// TwinCAT 3 PLC project IoT_OPCUA
// ProgramVersion: 3.1.4023.0
// libraries:
//   Tc2_EtherCAT, * (Beckhoff Automation GmbH)
//   Tc2_MDP, * (Beckhoff Automation GmbH)
//   Tc2_ModbusSrv, * (Beckhoff Automation GmbH)
//   Tc2_Standard, * (Beckhoff Automation GmbH)
//   Tc2_System, * (Beckhoff Automation GmbH)
//   Tc2_Utilities, * (Beckhoff Automation GmbH)
//   Tc3_IPCDiag, * (Beckhoff Automation GmbH)
//   Tc3_Module, * (Beckhoff Automation GmbH)
//   BASIC,3.31,OSCAT
//   Tc2_OpcUa,3.3.2.0,Beckhoff Automation GmbH
//   VisuSymbols,3.5.10.0,System
// project tree:
//   / Class Diagram.TcCD (not stored), GlobalTextList.TcGTLO, PlcTask_10ms.TcTTO, PlcTask_500us.TcTTO, Task_1ms.TcTTO, Visualization Manager.TcVMO (not stored)
//   DUTs/ AirValveSimSignals.TcDUT, ElectrDataModbusTCP.TcDUT, ElectrDataEthCAT.TcDUT
//   DUTs/DataModels/ DriveState_DataModel.TcDUT, ElectrDevicePeriodicOper_DataModel.TcDUT, ElectrDeviceContOper_DataModel.TcDUT, SingleSensor_DataModel.TcDUT, SingleState_DataModel.TcDUT, ValveTravelTime_DataModel.TcDUT, VibAccelarationDataModel.TcDUT
//   GVLs/ GVL_const.TcGVL, GVL_SW.TcGVL, GVL_HW.TcGVL, GVL_Visu.TcGVL
//   POUs/EL3443/EL3443/DUTs/ E_EL3443_Phase.TcDUT, E_EL3443_Total.TcDUT, ST_EL3443_MUX_REAL.TcDUT, ST_EL3443_MUX_ULINT.TcDUT, ST_EL3443_StatusLx.TcDUT, ST_EL3443_StatusTotal.TcDUT, ST_EL3443_VariantLx.TcDUT, ST_EL3443_VariantTotal.TcDUT, ST_EL3443_VariantValues.TcDUT
//   POUs/EL3443/EL3443/ FB_EL3443.TcPOU (not stored)
//   POUs/EL3443/EL3443_DPM/DUTs/ E_EL3443_DPM_Phase.TcDUT, E_EL3443_DPM_Total.TcDUT, ST_EL3443_DPM_MUX_REAL.TcDUT, ST_EL3443_DPM_MUX_ULINT.TcDUT, ST_EL3443_DPM_StatusLx.TcDUT, ST_EL3443_DPM_StatusTotal.TcDUT, ST_EL3443_DPM_VariantLx.TcDUT, ST_EL3443_DPM_VariantTotal.TcDUT, ST_EL3443_DPM_VariantValues.TcDUT
//   POUs/EL3443/EL3443_DPM/ FB_EL3443_DPM.TcPOU
//   POUs/FB/Generic/ CheckLineProducing.TcPOU, PartsPerMinHistorical.TcPOU, PartsPerMinInstant.TcPOU, PartsPerMinInstant2.TcPOU, ReadMemoryUsage.TcPOU, Valve_Signal_Sim.TcPOU, TONR.TcPOU, UnixTimestamp.TcPOU, ValueChangeDetector.TcPOU
//   POUs/FB/ModbusTCP/ ReadMBSentron_PAC1200.TcPOU
//   POUs/FB/OPC_UA/ ElectricalDevicePeriodicOper.TcPOU, ElectricalDeviceContOper.TcPOU, GenericSensor.TcPOU, GenericState.TcPOU, Valve2Cmd2FB.TcPOU, VibrationSensor.TcPOU
//   POUs/FC/ AI_Scale.TcPOU
//   POUs/PRG_10ms/ PRG_06_ElectricalMonitoring.TcPOU, PRG_04_AirValveAnalytics.TcPOU, PRG_05_ElectricalAnalytics.TcPOU, PRG_01_MAIN.TcPOU, PRG_09_PlcDiagnostic.TcPOU, PRG_08_ProductionStatistics.TcPOU, PRG_10_TempHumidAnalytics.TcPOU, PRG_11_AirFlowAnalytics.TcPOU, PRG_12_OilContaminationAnalytics.TcPOU, Simulation.TcPOU, PRG_02_DataMapping.TcPOU, PRG_07_LineState.TcPOU, PRG_03_VibrationAnalytics.TcPOU
//   POUs/PRG_1ms/ Main_T1ms.TcPOU, TimeStamp.TcPOU
//   POUs/PRG_500us/ Main_500us.TcPOU
//   VISU/ TextList1.TcTLO, Visualization1.TcVIS
// real-time tasks:
//   TASK PlcTask_10ms: cycle T#10ms, priority 20, ADS port 350
//   TASK Task_1ms: cycle T#1ms, priority 1, ADS port 351
//   TASK ProfiNET: cycle T#2ms, priority 2, ADS port 301
//   TASK PlcTask_500us: cycle T#500us, priority 23, ADS port 354
// I/O:
//   DEVICE Device1 (Profinet Device) (disabled), AmsNetId 192.168.149.130.2.1
//     profinet-io-device [Beckhoff Automation TwinCAT PLC PROFINET I/O Device with I/Os, V2.32, 1 port diagnostic supported TwinCAT PN Device]
//       modules: Term 1 (DAP Module), Term 2 (32 Word Output), Term 3 (32 DWord Output), Term 4 (10 Float32 Output), Term 5 (10 Float32 Input)
//   DEVICE Device2 (EtherCAT) (disabled), AmsNetId 192.168.149.130.3.1
//     ElectricalCabinet [EK1100 EtherCAT Coupler (2A E-Bus)]
//       Term_1 (EL3443) [EL3443 3Ch. Power Measuring]
//       Term_2 (EL3443) [EL3443 3Ch. Power Measuring]
//       Term_3 (EL3152) [EL3152 2Ch. Ana Input 4-20mA]
//       Term_4 (EL6601) [EL6601 1 Port Switch (Ethernet, CoE)]
//       Term_99 (EL9011) [EL9011 End Terminal]
//     IO_LinkNode1 (EP6228-0022) [EP6228-0022 (IO Link Master)]
//       modules: Module 1 (DeviceState Inputs Device), Module 2 (DeviceState Inputs), IoLinkNode1_Ch1 (IO-Link Slave), IoLinkNode1_Ch2 (IO-Link Slave), IoLinkNode1_Ch3 (IO-Link Slave), IoLinkNode1_Ch4 (IO-Link Slave), IoLinkNode1_Ch5 (IO-Link Slave), IoLinkNode1_Ch6 (IO-Link Slave), Module 9 (empty), Module 10 (empty)
//     IO_LinkNode2 (EP6224-2022) [EP6224-2022 (IO Link Master)]
//       modules: Module 1 (DeviceState Inputs Device), Module 2 (DeviceState Inputs), IoLinkNode2_Ch1 (IO-Link Slave), IoLinkNode2_Ch2 (IO-Link Slave), IoLinkNode2_Ch3 (IO-Link Slave), IoLinkNode2_Ch4 (IO-Link Slave)
//   DEVICE Device 3 (USB) (disabled)
//     Box 2 (C9900-L100 License-Key-USB-Stick)
// variable links:
//   IoT_OPCUA/IoT_OPCUA Instance <-> Device1 (Profinet Device)/profinet-io-device
//     PlcTask_10ms Inputs/GVL_HW.PnIoDevice_10Real_In <-> API/Term 4 (10 Float32 Output)/Subterm 6 (10 Float32 Output)/Inputs/1 Float32 Output[0]
//     PlcTask_10ms Inputs/GVL_HW.PnIoDevice_10Real_In @bit {32..288 step 32} <-> API/Term 4 (10 Float32 Output)/Subterm 6 (10 Float32 Output)/Inputs/1 Float32 Output[{1..9}]  (9 links)
//     PlcTask_10ms Inputs/GVL_HW.PnIoDevice_32DWord_In <-> API/Term 3 (32 DWord Output)/Subterm 5 (32 DWord Output)/Inputs/1 DWord Output[0]
//     PlcTask_10ms Inputs/GVL_HW.PnIoDevice_32DWord_In @bit {32..992 step 32} <-> API/Term 3 (32 DWord Output)/Subterm 5 (32 DWord Output)/Inputs/1 DWord Output[{1..31}]  (31 links)
//     PlcTask_10ms Inputs/GVL_HW.PnIoDevice_32Word_In <-> API/Term 2 (32 Word Output)/Subterm 4 (32 Word Output)/Inputs/1 Word Output[0]
//     PlcTask_10ms Inputs/GVL_HW.PnIoDevice_32Word_In @bit {16..496 step 16} <-> API/Term 2 (32 Word Output)/Subterm 4 (32 Word Output)/Inputs/1 Word Output[{1..31}]  (31 links)
//     PlcTask_10ms Outputs/GVL_HW.PnIoDevice_10Real_Out <-> API/Term 5 (10 Float32 Input)/Subterm 7 (10 Float32 Input)/Outputs/1 Float32 Input[0]
//     PlcTask_10ms Outputs/GVL_HW.PnIoDevice_10Real_Out @bit {32..288 step 32} <-> API/Term 5 (10 Float32 Input)/Subterm 7 (10 Float32 Input)/Outputs/1 Float32 Input[{1..9}]  (9 links)
//   IoT_OPCUA/IoT_OPCUA Instance <-> Device2 (EtherCAT)/ElectricalCabinet/Term_1 (EL3443)
//     PlcTask_500us Inputs/Main_500us.ElectricalDevice1.stEL3443_IO.MDP5001_341_Input/MDP5001_341_L1_Basic_Current <-> L1 Basic/Current
//     PlcTask_500us Inputs/Main_500us.ElectricalDevice1.stEL3443_IO.MDP5001_341_Input/MDP5001_341_L2_Basic_Current <-> L2 Basic/Current
//     PlcTask_500us Inputs/Main_500us.ElectricalDevice1.stEL3443_IO.MDP5001_341_Input/MDP5001_341_L3_Basic_Current <-> L3 Basic/Current
//     PlcTask_500us Inputs/Main_500us.ElectricalDevice1.stEL3443_IO.MDP5001_341_Input/MDP5001_341_L1_Basic_Voltage <-> L1 Basic/Voltage
//     PlcTask_500us Inputs/Main_500us.ElectricalDevice1.stEL3443_IO.MDP5001_341_Input/MDP5001_341_L2_Basic_Voltage <-> L2 Basic/Voltage
//     PlcTask_500us Inputs/Main_500us.ElectricalDevice1.stEL3443_IO.MDP5001_341_Input/MDP5001_341_L3_Basic_Voltage <-> L3 Basic/Voltage
//     PlcTask_500us Inputs/Main_500us.ElectricalDevice1.stEL3443_IO.MDP5001_341_Input/MDP5001_341_L1_Power_Active_Power <-> L1 Power/Active Power
//     PlcTask_500us Inputs/Main_500us.ElectricalDevice1.stEL3443_IO.MDP5001_341_Input/MDP5001_341_L2_Power_Active_Power <-> L2 Power/Active Power
//     PlcTask_500us Inputs/Main_500us.ElectricalDevice1.stEL3443_IO.MDP5001_341_Input/MDP5001_341_L3_Power_Active_Power <-> L3 Power/Active Power
//     PlcTask_500us Inputs/Main_500us.ElectricalDevice1.stEL3443_IO.MDP5001_341_Input/MDP5001_341_L1_Power_Apparent_Power <-> L1 Power/Apparent Power
//     PlcTask_500us Inputs/Main_500us.ElectricalDevice1.stEL3443_IO.MDP5001_341_Input/MDP5001_341_L2_Power_Apparent_Power <-> L2 Power/Apparent Power
//     PlcTask_500us Inputs/Main_500us.ElectricalDevice1.stEL3443_IO.MDP5001_341_Input/MDP5001_341_L3_Power_Apparent_Power <-> L3 Power/Apparent Power
//     PlcTask_500us Inputs/Main_500us.ElectricalDevice1.stEL3443_IO.MDP5001_341_Input/MDP5001_341_L1_Power_Power_Factor <-> L1 Power/Power Factor
//     PlcTask_500us Inputs/Main_500us.ElectricalDevice1.stEL3443_IO.MDP5001_341_Input/MDP5001_341_L2_Power_Power_Factor <-> L2 Power/Power Factor
//     PlcTask_500us Inputs/Main_500us.ElectricalDevice1.stEL3443_IO.MDP5001_341_Input/MDP5001_341_L3_Power_Power_Factor <-> L3 Power/Power Factor
//     PlcTask_500us Inputs/Main_500us.ElectricalDevice1.stEL3443_IO.MDP5001_341_Input/MDP5001_341_L1_Power_Reactive_Power <-> L1 Power/Reactive Power
//     PlcTask_500us Inputs/Main_500us.ElectricalDevice1.stEL3443_IO.MDP5001_341_Input/MDP5001_341_L2_Power_Reactive_Power <-> L2 Power/Reactive Power
//     PlcTask_500us Inputs/Main_500us.ElectricalDevice1.stEL3443_IO.MDP5001_341_Input/MDP5001_341_L3_Power_Reactive_Power <-> L3 Power/Reactive Power
//     PlcTask_500us Inputs/Main_500us.ElectricalDevice1.stEL3443_IO.MDP5001_341_Input/MDP5001_341_L1_Status_Current_Guard_Error <-> L1 Status/Current Guard Error
//     PlcTask_500us Inputs/Main_500us.ElectricalDevice1.stEL3443_IO.MDP5001_341_Input/MDP5001_341_L2_Status_Current_Guard_Error <-> L2 Status/Current Guard Error
//     PlcTask_500us Inputs/Main_500us.ElectricalDevice1.stEL3443_IO.MDP5001_341_Input/MDP5001_341_L3_Status_Current_Guard_Error <-> L3 Status/Current Guard Error
//     PlcTask_500us Inputs/Main_500us.ElectricalDevice1.stEL3443_IO.MDP5001_341_Input/MDP5001_341_L1_Status_Current_Guard_Warning <-> L1 Status/Current Guard Warning
//     PlcTask_500us Inputs/Main_500us.ElectricalDevice1.stEL3443_IO.MDP5001_341_Input/MDP5001_341_L2_Status_Current_Guard_Warning <-> L2 Status/Current Guard Warning
//     PlcTask_500us Inputs/Main_500us.ElectricalDevice1.stEL3443_IO.MDP5001_341_Input/MDP5001_341_L3_Status_Current_Guard_Warning <-> L3 Status/Current Guard Warning
//     PlcTask_500us Inputs/Main_500us.ElectricalDevice1.stEL3443_IO.MDP5001_341_Input/MDP5001_341_L1_Status_Inaccurate_Current <-> L1 Status/Inaccurate Current
//     PlcTask_500us Inputs/Main_500us.ElectricalDevice1.stEL3443_IO.MDP5001_341_Input/MDP5001_341_L2_Status_Inaccurate_Current <-> L2 Status/Inaccurate Current
//     PlcTask_500us Inputs/Main_500us.ElectricalDevice1.stEL3443_IO.MDP5001_341_Input/MDP5001_341_L3_Status_Inaccurate_Current <-> L3 Status/Inaccurate Current
//     PlcTask_500us Inputs/Main_500us.ElectricalDevice1.stEL3443_IO.MDP5001_341_Input/MDP5001_341_L1_Status_Inaccurate_Voltage <-> L1 Status/Inaccurate Voltage
//     PlcTask_500us Inputs/Main_500us.ElectricalDevice1.stEL3443_IO.MDP5001_341_Input/MDP5001_341_L2_Status_Inaccurate_Voltage <-> L2 Status/Inaccurate Voltage
//     PlcTask_500us Inputs/Main_500us.ElectricalDevice1.stEL3443_IO.MDP5001_341_Input/MDP5001_341_L3_Status_Inaccurate_Voltage <-> L3 Status/Inaccurate Voltage
//     PlcTask_500us Inputs/Main_500us.ElectricalDevice1.stEL3443_IO.MDP5001_341_Input/MDP5001_341_L1_Status_Overcurrent <-> L1 Status/Overcurrent
//     PlcTask_500us Inputs/Main_500us.ElectricalDevice1.stEL3443_IO.MDP5001_341_Input/MDP5001_341_L2_Status_Overcurrent <-> L2 Status/Overcurrent
//     PlcTask_500us Inputs/Main_500us.ElectricalDevice1.stEL3443_IO.MDP5001_341_Input/MDP5001_341_L3_Status_Overcurrent <-> L3 Status/Overcurrent
//     PlcTask_500us Inputs/Main_500us.ElectricalDevice1.stEL3443_IO.MDP5001_341_Input/MDP5001_341_L1_Status_Overvoltage <-> L1 Status/Overvoltage
//     PlcTask_500us Inputs/Main_500us.ElectricalDevice1.stEL3443_IO.MDP5001_341_Input/MDP5001_341_L2_Status_Overvoltage <-> L2 Status/Overvoltage
//     PlcTask_500us Inputs/Main_500us.ElectricalDevice1.stEL3443_IO.MDP5001_341_Input/MDP5001_341_L3_Status_Overvoltage <-> L3 Status/Overvoltage
//     PlcTask_500us Inputs/Main_500us.ElectricalDevice1.stEL3443_IO.MDP5001_341_Input/MDP5001_341_L1_Status_TxPDO_Toggle <-> L1 Status/TxPDO Toggle
//     PlcTask_500us Inputs/Main_500us.ElectricalDevice1.stEL3443_IO.MDP5001_341_Input/MDP5001_341_L2_Status_TxPDO_Toggle <-> L2 Status/TxPDO Toggle
//     PlcTask_500us Inputs/Main_500us.ElectricalDevice1.stEL3443_IO.MDP5001_341_Input/MDP5001_341_L3_Status_TxPDO_Toggle <-> L3 Status/TxPDO Toggle
//     PlcTask_500us Inputs/Main_500us.ElectricalDevice1.stEL3443_IO.MDP5001_341_Input/MDP5001_341_L1_Status_Voltage_Guard_Error <-> L1 Status/Voltage Guard Error
//     PlcTask_500us Inputs/Main_500us.ElectricalDevice1.stEL3443_IO.MDP5001_341_Input/MDP5001_341_L2_Status_Voltage_Guard_Error <-> L2 Status/Voltage Guard Error
//     PlcTask_500us Inputs/Main_500us.ElectricalDevice1.stEL3443_IO.MDP5001_341_Input/MDP5001_341_L3_Status_Voltage_Guard_Error <-> L3 Status/Voltage Guard Error
//     PlcTask_500us Inputs/Main_500us.ElectricalDevice1.stEL3443_IO.MDP5001_341_Input/MDP5001_341_L1_Status_Voltage_Guard_Warning <-> L1 Status/Voltage Guard Warning
//     PlcTask_500us Inputs/Main_500us.ElectricalDevice1.stEL3443_IO.MDP5001_341_Input/MDP5001_341_L2_Status_Voltage_Guard_Warning <-> L2 Status/Voltage Guard Warning
//     PlcTask_500us Inputs/Main_500us.ElectricalDevice1.stEL3443_IO.MDP5001_341_Input/MDP5001_341_L3_Status_Voltage_Guard_Warning <-> L3 Status/Voltage Guard Warning
//     PlcTask_500us Inputs/Main_500us.ElectricalDevice1.stEL3443_IO.MDP5001_341_Input/MDP5001_341_L1_Status_Voltage_Sign_Bit <-> L1 Status/Voltage Sign Bit
//     PlcTask_500us Inputs/Main_500us.ElectricalDevice1.stEL3443_IO.MDP5001_341_Input/MDP5001_341_L2_Status_Voltage_Sign_Bit <-> L2 Status/Voltage Sign Bit
//     PlcTask_500us Inputs/Main_500us.ElectricalDevice1.stEL3443_IO.MDP5001_341_Input/MDP5001_341_L3_Status_Voltage_Sign_Bit <-> L3 Status/Voltage Sign Bit
//     PlcTask_500us Inputs/Main_500us.ElectricalDevice1.stEL3443_IO.MDP5001_341_Input/MDP5001_341_L1_Timing_Voltage_Last_Zero_Crossing <-> L1 Timing/Voltage Last Zero Crossing
//     PlcTask_500us Inputs/Main_500us.ElectricalDevice1.stEL3443_IO.MDP5001_341_Input/MDP5001_341_L2_Timing_Voltage_Last_Zero_Crossing <-> L2 Timing/Voltage Last Zero Crossing
//     PlcTask_500us Inputs/Main_500us.ElectricalDevice1.stEL3443_IO.MDP5001_341_Input/MDP5001_341_L3_Timing_Voltage_Last_Zero_Crossing <-> L3 Timing/Voltage Last Zero Crossing
//     PlcTask_500us Inputs/Main_500us.ElectricalDevice1.stEL3443_IO.MDP5001_341_Input/MDP5001_341_Total_Basic_Calculated_Neutral_Line_Current <-> Total Basic/Calculated Neutral Line Current
//     PlcTask_500us Inputs/Main_500us.ElectricalDevice1.stEL3443_IO.MDP5001_341_Input/MDP5001_341_Total_Basic_Frequency <-> Total Basic/Frequency
//     PlcTask_500us Inputs/Main_500us.ElectricalDevice1.stEL3443_IO.MDP5001_341_Input/MDP5001_341_Total_Basic_Power_Factor <-> Total Basic/Power Factor
//     PlcTask_500us Inputs/Main_500us.ElectricalDevice1.stEL3443_IO.MDP5001_341_Input/MDP5001_341_Total_Status_Active_Power_Guard_Error <-> Total Status/Active Power Guard Error
//     PlcTask_500us Inputs/Main_500us.ElectricalDevice1.stEL3443_IO.MDP5001_341_Input/MDP5001_341_Total_Status_Active_Power_Guard_Warning <-> Total Status/Active Power Guard Warning
//     PlcTask_500us Inputs/Main_500us.ElectricalDevice1.stEL3443_IO.MDP5001_341_Input/MDP5001_341_Total_Status_Apparent_Power_Guard_Error <-> Total Status/Apparent Power Guard Error
//     PlcTask_500us Inputs/Main_500us.ElectricalDevice1.stEL3443_IO.MDP5001_341_Input/MDP5001_341_Total_Status_Apparent_Power_Guard_Warning <-> Total Status/Apparent Power Guard Warning
//     PlcTask_500us Inputs/Main_500us.ElectricalDevice1.stEL3443_IO.MDP5001_341_Input/MDP5001_341_Total_Status_Frequency_Guard_Error <-> Total Status/Frequency Guard Error
//     PlcTask_500us Inputs/Main_500us.ElectricalDevice1.stEL3443_IO.MDP5001_341_Input/MDP5001_341_Total_Status_Frequency_Guard_Warning <-> Total Status/Frequency Guard Warning
//     PlcTask_500us Inputs/Main_500us.ElectricalDevice1.stEL3443_IO.MDP5001_341_Input/MDP5001_341_Total_Status_Grid_Direction <-> Total Status/Grid Direction
//     PlcTask_500us Inputs/Main_500us.ElectricalDevice1.stEL3443_IO.MDP5001_341_Input/MDP5001_341_Total_Status_Neutral_Current_Guard_Error <-> Total Status/Neutral Current Guard Error
//     PlcTask_500us Inputs/Main_500us.ElectricalDevice1.stEL3443_IO.MDP5001_341_Input/MDP5001_341_Total_Status_Neutral_Current_Guard_Warning <-> Total Status/Neutral Current Guard Warning
//     PlcTask_500us Inputs/Main_500us.ElectricalDevice1.stEL3443_IO.MDP5001_341_Input/MDP5001_341_Total_Status_Power_Quality_Factor <-> Total Status/Power Quality Factor
//     PlcTask_500us Inputs/Main_500us.ElectricalDevice1.stEL3443_IO.MDP5001_341_Input/MDP5001_341_Total_Status_Power_Quality_Guard_Error <-> Total Status/Power Quality Guard Error
//     PlcTask_500us Inputs/Main_500us.ElectricalDevice1.stEL3443_IO.MDP5001_341_Input/MDP5001_341_Total_Status_Power_Quality_Guard_Warning <-> Total Status/Power Quality Guard Warning
//     PlcTask_500us Inputs/Main_500us.ElectricalDevice1.stEL3443_IO.MDP5001_341_Input/MDP5001_341_Total_Status_System_State <-> Total Status/System State
//     PlcTask_500us Inputs/Main_500us.ElectricalDevice1.stEL3443_IO.MDP5001_341_Input/MDP5001_341_Total_Status_TxPDO_State <-> Total Status/TxPDO State
//     PlcTask_500us Inputs/Main_500us.ElectricalDevice1.stEL3443_IO.MDP5001_341_Input/MDP5001_341_Total_Status_TxPDO_Toggle <-> Total Status/TxPDO Toggle
//     PlcTask_500us Inputs/Main_500us.ElectricalDevice1.stEL3443_IO.MDP5001_341_Input/MDP5001_341_Total_Variant_Value_In_Index_1_REAL <-> Total Variant Value In/Index 1 REAL
//     PlcTask_500us Inputs/Main_500us.ElectricalDevice1.stEL3443_IO.MDP5001_341_Input/MDP5001_341_Total_Variant_Value_In_Index_2_REAL <-> Total Variant Value In/Index 2 REAL
//     PlcTask_500us Inputs/Main_500us.ElectricalDevice1.stEL3443_IO.MDP5001_341_Input/MDP5001_341_Total_Variant_Value_In_Index_3_REAL <-> Total Variant Value In/Index 3 REAL
//     PlcTask_500us Inputs/Main_500us.ElectricalDevice1.stEL3443_IO.MDP5001_341_Input/MDP5001_341_Total_Variant_Value_In_Index_4_ULINT <-> Total Variant Value In/Index 4 ULINT
//     PlcTask_500us Inputs/Main_500us.ElectricalDevice1.stEL3443_IO.MDP5001_341_Input/MDP5001_341_Total_Variant_Value_In_TxPDO_Toggle <-> Total Variant Value In/TxPDO Toggle
//     PlcTask_500us Inputs/Main_500us.ElectricalDevice1.stEL3443_IO.MDP5001_341_Input/MDP5001_341_Total_Variant_Value_In_Value_1_REAL <-> Total Variant Value In/Value 1 REAL
//     PlcTask_500us Inputs/Main_500us.ElectricalDevice1.stEL3443_IO.MDP5001_341_Input/MDP5001_341_Total_Variant_Value_In_Value_2_REAL <-> Total Variant Value In/Value 2 REAL
//     PlcTask_500us Inputs/Main_500us.ElectricalDevice1.stEL3443_IO.MDP5001_341_Input/MDP5001_341_Total_Variant_Value_In_Value_3_REAL <-> Total Variant Value In/Value 3 REAL
//     PlcTask_500us Inputs/Main_500us.ElectricalDevice1.stEL3443_IO.MDP5001_341_Input/MDP5001_341_Total_Variant_Value_In_Value_4_ULINT <-> Total Variant Value In/Value 4 ULINT
//     PlcTask_500us Outputs/Main_500us.ElectricalDevice1.stEL3443_IO.MDP5001_341_Output/MDP5001_341_Total_Variant_Value_Out_Index_1_REAL <-> Total Variant Value Out/Index 1 REAL
//     PlcTask_500us Outputs/Main_500us.ElectricalDevice1.stEL3443_IO.MDP5001_341_Output/MDP5001_341_Total_Variant_Value_Out_Index_2_REAL <-> Total Variant Value Out/Index 2 REAL
//     PlcTask_500us Outputs/Main_500us.ElectricalDevice1.stEL3443_IO.MDP5001_341_Output/MDP5001_341_Total_Variant_Value_Out_Index_3_REAL <-> Total Variant Value Out/Index 3 REAL
//     PlcTask_500us Outputs/Main_500us.ElectricalDevice1.stEL3443_IO.MDP5001_341_Output/MDP5001_341_Total_Variant_Value_Out_Index_4_ULINT <-> Total Variant Value Out/Index 4 ULINT
//   IoT_OPCUA/IoT_OPCUA Instance <-> Device2 (EtherCAT)/ElectricalCabinet/Term_2 (EL3443)
//     PlcTask_500us Inputs/Main_500us.ElectricalDevice2.stEL3443_IO.MDP5001_341_Input/MDP5001_341_L1_Basic_Current <-> L1 Basic/Current
//     PlcTask_500us Inputs/Main_500us.ElectricalDevice2.stEL3443_IO.MDP5001_341_Input/MDP5001_341_L2_Basic_Current <-> L2 Basic/Current
//     PlcTask_500us Inputs/Main_500us.ElectricalDevice2.stEL3443_IO.MDP5001_341_Input/MDP5001_341_L3_Basic_Current <-> L3 Basic/Current
//     PlcTask_500us Inputs/Main_500us.ElectricalDevice2.stEL3443_IO.MDP5001_341_Input/MDP5001_341_L1_Basic_Voltage <-> L1 Basic/Voltage
//     PlcTask_500us Inputs/Main_500us.ElectricalDevice2.stEL3443_IO.MDP5001_341_Input/MDP5001_341_L2_Basic_Voltage <-> L2 Basic/Voltage
//     PlcTask_500us Inputs/Main_500us.ElectricalDevice2.stEL3443_IO.MDP5001_341_Input/MDP5001_341_L3_Basic_Voltage <-> L3 Basic/Voltage
//     PlcTask_500us Inputs/Main_500us.ElectricalDevice2.stEL3443_IO.MDP5001_341_Input/MDP5001_341_L1_Power_Active_Power <-> L1 Power/Active Power
//     PlcTask_500us Inputs/Main_500us.ElectricalDevice2.stEL3443_IO.MDP5001_341_Input/MDP5001_341_L2_Power_Active_Power <-> L2 Power/Active Power
//     PlcTask_500us Inputs/Main_500us.ElectricalDevice2.stEL3443_IO.MDP5001_341_Input/MDP5001_341_L3_Power_Active_Power <-> L3 Power/Active Power
//     PlcTask_500us Inputs/Main_500us.ElectricalDevice2.stEL3443_IO.MDP5001_341_Input/MDP5001_341_L1_Power_Apparent_Power <-> L1 Power/Apparent Power
//     PlcTask_500us Inputs/Main_500us.ElectricalDevice2.stEL3443_IO.MDP5001_341_Input/MDP5001_341_L2_Power_Apparent_Power <-> L2 Power/Apparent Power
//     PlcTask_500us Inputs/Main_500us.ElectricalDevice2.stEL3443_IO.MDP5001_341_Input/MDP5001_341_L3_Power_Apparent_Power <-> L3 Power/Apparent Power
//     PlcTask_500us Inputs/Main_500us.ElectricalDevice2.stEL3443_IO.MDP5001_341_Input/MDP5001_341_L1_Power_Power_Factor <-> L1 Power/Power Factor
//     PlcTask_500us Inputs/Main_500us.ElectricalDevice2.stEL3443_IO.MDP5001_341_Input/MDP5001_341_L2_Power_Power_Factor <-> L2 Power/Power Factor
//     PlcTask_500us Inputs/Main_500us.ElectricalDevice2.stEL3443_IO.MDP5001_341_Input/MDP5001_341_L3_Power_Power_Factor <-> L3 Power/Power Factor
//     PlcTask_500us Inputs/Main_500us.ElectricalDevice2.stEL3443_IO.MDP5001_341_Input/MDP5001_341_L1_Power_Reactive_Power <-> L1 Power/Reactive Power
//     PlcTask_500us Inputs/Main_500us.ElectricalDevice2.stEL3443_IO.MDP5001_341_Input/MDP5001_341_L2_Power_Reactive_Power <-> L2 Power/Reactive Power
//     PlcTask_500us Inputs/Main_500us.ElectricalDevice2.stEL3443_IO.MDP5001_341_Input/MDP5001_341_L3_Power_Reactive_Power <-> L3 Power/Reactive Power
//     PlcTask_500us Inputs/Main_500us.ElectricalDevice2.stEL3443_IO.MDP5001_341_Input/MDP5001_341_L1_Status_Current_Guard_Error <-> L1 Status/Current Guard Error
//     PlcTask_500us Inputs/Main_500us.ElectricalDevice2.stEL3443_IO.MDP5001_341_Input/MDP5001_341_L2_Status_Current_Guard_Error <-> L2 Status/Current Guard Error
//     PlcTask_500us Inputs/Main_500us.ElectricalDevice2.stEL3443_IO.MDP5001_341_Input/MDP5001_341_L3_Status_Current_Guard_Error <-> L3 Status/Current Guard Error
//     PlcTask_500us Inputs/Main_500us.ElectricalDevice2.stEL3443_IO.MDP5001_341_Input/MDP5001_341_L1_Status_Current_Guard_Warning <-> L1 Status/Current Guard Warning
//     PlcTask_500us Inputs/Main_500us.ElectricalDevice2.stEL3443_IO.MDP5001_341_Input/MDP5001_341_L2_Status_Current_Guard_Warning <-> L2 Status/Current Guard Warning
//     PlcTask_500us Inputs/Main_500us.ElectricalDevice2.stEL3443_IO.MDP5001_341_Input/MDP5001_341_L3_Status_Current_Guard_Warning <-> L3 Status/Current Guard Warning
//     PlcTask_500us Inputs/Main_500us.ElectricalDevice2.stEL3443_IO.MDP5001_341_Input/MDP5001_341_L1_Status_Inaccurate_Current <-> L1 Status/Inaccurate Current
//     PlcTask_500us Inputs/Main_500us.ElectricalDevice2.stEL3443_IO.MDP5001_341_Input/MDP5001_341_L2_Status_Inaccurate_Current <-> L2 Status/Inaccurate Current
//     PlcTask_500us Inputs/Main_500us.ElectricalDevice2.stEL3443_IO.MDP5001_341_Input/MDP5001_341_L3_Status_Inaccurate_Current <-> L3 Status/Inaccurate Current
//     PlcTask_500us Inputs/Main_500us.ElectricalDevice2.stEL3443_IO.MDP5001_341_Input/MDP5001_341_L1_Status_Inaccurate_Voltage <-> L1 Status/Inaccurate Voltage
//     PlcTask_500us Inputs/Main_500us.ElectricalDevice2.stEL3443_IO.MDP5001_341_Input/MDP5001_341_L2_Status_Inaccurate_Voltage <-> L2 Status/Inaccurate Voltage
//     PlcTask_500us Inputs/Main_500us.ElectricalDevice2.stEL3443_IO.MDP5001_341_Input/MDP5001_341_L3_Status_Inaccurate_Voltage <-> L3 Status/Inaccurate Voltage
//     PlcTask_500us Inputs/Main_500us.ElectricalDevice2.stEL3443_IO.MDP5001_341_Input/MDP5001_341_L1_Status_Overcurrent <-> L1 Status/Overcurrent
//     PlcTask_500us Inputs/Main_500us.ElectricalDevice2.stEL3443_IO.MDP5001_341_Input/MDP5001_341_L2_Status_Overcurrent <-> L2 Status/Overcurrent
//     PlcTask_500us Inputs/Main_500us.ElectricalDevice2.stEL3443_IO.MDP5001_341_Input/MDP5001_341_L3_Status_Overcurrent <-> L3 Status/Overcurrent
//     PlcTask_500us Inputs/Main_500us.ElectricalDevice2.stEL3443_IO.MDP5001_341_Input/MDP5001_341_L1_Status_Overvoltage <-> L1 Status/Overvoltage
//     PlcTask_500us Inputs/Main_500us.ElectricalDevice2.stEL3443_IO.MDP5001_341_Input/MDP5001_341_L2_Status_Overvoltage <-> L2 Status/Overvoltage
//     PlcTask_500us Inputs/Main_500us.ElectricalDevice2.stEL3443_IO.MDP5001_341_Input/MDP5001_341_L3_Status_Overvoltage <-> L3 Status/Overvoltage
//     PlcTask_500us Inputs/Main_500us.ElectricalDevice2.stEL3443_IO.MDP5001_341_Input/MDP5001_341_L1_Status_TxPDO_Toggle <-> L1 Status/TxPDO Toggle
//     PlcTask_500us Inputs/Main_500us.ElectricalDevice2.stEL3443_IO.MDP5001_341_Input/MDP5001_341_L2_Status_TxPDO_Toggle <-> L2 Status/TxPDO Toggle
//     PlcTask_500us Inputs/Main_500us.ElectricalDevice2.stEL3443_IO.MDP5001_341_Input/MDP5001_341_L3_Status_TxPDO_Toggle <-> L3 Status/TxPDO Toggle
//     PlcTask_500us Inputs/Main_500us.ElectricalDevice2.stEL3443_IO.MDP5001_341_Input/MDP5001_341_L1_Status_Voltage_Guard_Error <-> L1 Status/Voltage Guard Error
//     PlcTask_500us Inputs/Main_500us.ElectricalDevice2.stEL3443_IO.MDP5001_341_Input/MDP5001_341_L2_Status_Voltage_Guard_Error <-> L2 Status/Voltage Guard Error
//     PlcTask_500us Inputs/Main_500us.ElectricalDevice2.stEL3443_IO.MDP5001_341_Input/MDP5001_341_L3_Status_Voltage_Guard_Error <-> L3 Status/Voltage Guard Error
//     PlcTask_500us Inputs/Main_500us.ElectricalDevice2.stEL3443_IO.MDP5001_341_Input/MDP5001_341_L1_Status_Voltage_Guard_Warning <-> L1 Status/Voltage Guard Warning
//     PlcTask_500us Inputs/Main_500us.ElectricalDevice2.stEL3443_IO.MDP5001_341_Input/MDP5001_341_L2_Status_Voltage_Guard_Warning <-> L2 Status/Voltage Guard Warning
//     PlcTask_500us Inputs/Main_500us.ElectricalDevice2.stEL3443_IO.MDP5001_341_Input/MDP5001_341_L3_Status_Voltage_Guard_Warning <-> L3 Status/Voltage Guard Warning
//     PlcTask_500us Inputs/Main_500us.ElectricalDevice2.stEL3443_IO.MDP5001_341_Input/MDP5001_341_L1_Status_Voltage_Sign_Bit <-> L1 Status/Voltage Sign Bit
//     PlcTask_500us Inputs/Main_500us.ElectricalDevice2.stEL3443_IO.MDP5001_341_Input/MDP5001_341_L2_Status_Voltage_Sign_Bit <-> L2 Status/Voltage Sign Bit
//     PlcTask_500us Inputs/Main_500us.ElectricalDevice2.stEL3443_IO.MDP5001_341_Input/MDP5001_341_L3_Status_Voltage_Sign_Bit <-> L3 Status/Voltage Sign Bit
//     PlcTask_500us Inputs/Main_500us.ElectricalDevice2.stEL3443_IO.MDP5001_341_Input/MDP5001_341_L1_Timing_Voltage_Last_Zero_Crossing <-> L1 Timing/Voltage Last Zero Crossing
//     PlcTask_500us Inputs/Main_500us.ElectricalDevice2.stEL3443_IO.MDP5001_341_Input/MDP5001_341_L2_Timing_Voltage_Last_Zero_Crossing <-> L2 Timing/Voltage Last Zero Crossing
//     PlcTask_500us Inputs/Main_500us.ElectricalDevice2.stEL3443_IO.MDP5001_341_Input/MDP5001_341_L3_Timing_Voltage_Last_Zero_Crossing <-> L3 Timing/Voltage Last Zero Crossing
//     PlcTask_500us Inputs/Main_500us.ElectricalDevice2.stEL3443_IO.MDP5001_341_Input/MDP5001_341_Total_Basic_Calculated_Neutral_Line_Current <-> Total Basic/Calculated Neutral Line Current
//     PlcTask_500us Inputs/Main_500us.ElectricalDevice2.stEL3443_IO.MDP5001_341_Input/MDP5001_341_Total_Basic_Frequency <-> Total Basic/Frequency
//     PlcTask_500us Inputs/Main_500us.ElectricalDevice2.stEL3443_IO.MDP5001_341_Input/MDP5001_341_Total_Basic_Power_Factor <-> Total Basic/Power Factor
//     PlcTask_500us Inputs/Main_500us.ElectricalDevice2.stEL3443_IO.MDP5001_341_Input/MDP5001_341_Total_Status_Active_Power_Guard_Error <-> Total Status/Active Power Guard Error
//     PlcTask_500us Inputs/Main_500us.ElectricalDevice2.stEL3443_IO.MDP5001_341_Input/MDP5001_341_Total_Status_Active_Power_Guard_Warning <-> Total Status/Active Power Guard Warning
//     PlcTask_500us Inputs/Main_500us.ElectricalDevice2.stEL3443_IO.MDP5001_341_Input/MDP5001_341_Total_Status_Apparent_Power_Guard_Error <-> Total Status/Apparent Power Guard Error
//     PlcTask_500us Inputs/Main_500us.ElectricalDevice2.stEL3443_IO.MDP5001_341_Input/MDP5001_341_Total_Status_Apparent_Power_Guard_Warning <-> Total Status/Apparent Power Guard Warning
//     PlcTask_500us Inputs/Main_500us.ElectricalDevice2.stEL3443_IO.MDP5001_341_Input/MDP5001_341_Total_Status_Frequency_Guard_Error <-> Total Status/Frequency Guard Error
//     PlcTask_500us Inputs/Main_500us.ElectricalDevice2.stEL3443_IO.MDP5001_341_Input/MDP5001_341_Total_Status_Frequency_Guard_Warning <-> Total Status/Frequency Guard Warning
//     PlcTask_500us Inputs/Main_500us.ElectricalDevice2.stEL3443_IO.MDP5001_341_Input/MDP5001_341_Total_Status_Grid_Direction <-> Total Status/Grid Direction
//     PlcTask_500us Inputs/Main_500us.ElectricalDevice2.stEL3443_IO.MDP5001_341_Input/MDP5001_341_Total_Status_Neutral_Current_Guard_Error <-> Total Status/Neutral Current Guard Error
//     PlcTask_500us Inputs/Main_500us.ElectricalDevice2.stEL3443_IO.MDP5001_341_Input/MDP5001_341_Total_Status_Neutral_Current_Guard_Warning <-> Total Status/Neutral Current Guard Warning
//     PlcTask_500us Inputs/Main_500us.ElectricalDevice2.stEL3443_IO.MDP5001_341_Input/MDP5001_341_Total_Status_Power_Quality_Factor <-> Total Status/Power Quality Factor
//     PlcTask_500us Inputs/Main_500us.ElectricalDevice2.stEL3443_IO.MDP5001_341_Input/MDP5001_341_Total_Status_Power_Quality_Guard_Error <-> Total Status/Power Quality Guard Error
//     PlcTask_500us Inputs/Main_500us.ElectricalDevice2.stEL3443_IO.MDP5001_341_Input/MDP5001_341_Total_Status_Power_Quality_Guard_Warning <-> Total Status/Power Quality Guard Warning
//     PlcTask_500us Inputs/Main_500us.ElectricalDevice2.stEL3443_IO.MDP5001_341_Input/MDP5001_341_Total_Status_System_State <-> Total Status/System State
//     PlcTask_500us Inputs/Main_500us.ElectricalDevice2.stEL3443_IO.MDP5001_341_Input/MDP5001_341_Total_Status_TxPDO_State <-> Total Status/TxPDO State
//     PlcTask_500us Inputs/Main_500us.ElectricalDevice2.stEL3443_IO.MDP5001_341_Input/MDP5001_341_Total_Status_TxPDO_Toggle <-> Total Status/TxPDO Toggle
//     PlcTask_500us Inputs/Main_500us.ElectricalDevice2.stEL3443_IO.MDP5001_341_Input/MDP5001_341_Total_Variant_Value_In_Index_1_REAL <-> Total Variant Value In/Index 1 REAL
//     PlcTask_500us Inputs/Main_500us.ElectricalDevice2.stEL3443_IO.MDP5001_341_Input/MDP5001_341_Total_Variant_Value_In_Index_2_REAL <-> Total Variant Value In/Index 2 REAL
//     PlcTask_500us Inputs/Main_500us.ElectricalDevice2.stEL3443_IO.MDP5001_341_Input/MDP5001_341_Total_Variant_Value_In_Index_3_REAL <-> Total Variant Value In/Index 3 REAL
//     PlcTask_500us Inputs/Main_500us.ElectricalDevice2.stEL3443_IO.MDP5001_341_Input/MDP5001_341_Total_Variant_Value_In_Index_4_ULINT <-> Total Variant Value In/Index 4 ULINT
//     PlcTask_500us Inputs/Main_500us.ElectricalDevice2.stEL3443_IO.MDP5001_341_Input/MDP5001_341_Total_Variant_Value_In_TxPDO_Toggle <-> Total Variant Value In/TxPDO Toggle
//     PlcTask_500us Inputs/Main_500us.ElectricalDevice2.stEL3443_IO.MDP5001_341_Input/MDP5001_341_Total_Variant_Value_In_Value_1_REAL <-> Total Variant Value In/Value 1 REAL
//     PlcTask_500us Inputs/Main_500us.ElectricalDevice2.stEL3443_IO.MDP5001_341_Input/MDP5001_341_Total_Variant_Value_In_Value_2_REAL <-> Total Variant Value In/Value 2 REAL
//     PlcTask_500us Inputs/Main_500us.ElectricalDevice2.stEL3443_IO.MDP5001_341_Input/MDP5001_341_Total_Variant_Value_In_Value_3_REAL <-> Total Variant Value In/Value 3 REAL
//     PlcTask_500us Inputs/Main_500us.ElectricalDevice2.stEL3443_IO.MDP5001_341_Input/MDP5001_341_Total_Variant_Value_In_Value_4_ULINT <-> Total Variant Value In/Value 4 ULINT
//     PlcTask_500us Outputs/Main_500us.ElectricalDevice2.stEL3443_IO.MDP5001_341_Output/MDP5001_341_Total_Variant_Value_Out_Index_1_REAL <-> Total Variant Value Out/Index 1 REAL
//     PlcTask_500us Outputs/Main_500us.ElectricalDevice2.stEL3443_IO.MDP5001_341_Output/MDP5001_341_Total_Variant_Value_Out_Index_2_REAL <-> Total Variant Value Out/Index 2 REAL
//     PlcTask_500us Outputs/Main_500us.ElectricalDevice2.stEL3443_IO.MDP5001_341_Output/MDP5001_341_Total_Variant_Value_Out_Index_3_REAL <-> Total Variant Value Out/Index 3 REAL
//     PlcTask_500us Outputs/Main_500us.ElectricalDevice2.stEL3443_IO.MDP5001_341_Output/MDP5001_341_Total_Variant_Value_Out_Index_4_ULINT <-> Total Variant Value Out/Index 4 ULINT
//   IoT_OPCUA/IoT_OPCUA Instance <-> Device2 (EtherCAT)/IO_LinkNode1 (EP6228-0022)
//     PlcTask_10ms Inputs/GVL_HW.IoLinkNode1Ch{1..6}_SensorTemp <-> IoLinkNode1_Ch{1..6} (IO-Link Slave)/IO-Link Port{1..6}/Contact Temperature Contact Temperature  (6 links)
//     PlcTask_10ms Inputs/GVL_HW.IoLinkNode1Ch{1..6}_VibAccelRmsX <-> IoLinkNode1_Ch{1..6} (IO-Link Slave)/IO-Link Port{1..6}/Vibration Acceleration RMS a-RMS X  (6 links)
//     PlcTask_10ms Inputs/GVL_HW.IoLinkNode1Ch{1..6}_VibAccelRmsY <-> IoLinkNode1_Ch{1..6} (IO-Link Slave)/IO-Link Port{1..6}/Vibration Acceleration RMS a-RMS Y  (6 links)
//     PlcTask_10ms Inputs/GVL_HW.IoLinkNode1Ch{1..6}_VibAccelRmsZ <-> IoLinkNode1_Ch{1..6} (IO-Link Slave)/IO-Link Port{1..6}/Vibration Acceleration RMS a-RMS Z  (6 links)
//   IoT_OPCUA/IoT_OPCUA Instance <-> Device2 (EtherCAT)/IO_LinkNode2 (EP6224-2022)
//     PlcTask_10ms Inputs/GVL_HW.IoLinkNode2Ch2_Humidity[1] <-> IoLinkNode2_Ch2 (IO-Link Slave)/IO-Link Port2/Port2: process data[3]
//     PlcTask_10ms Inputs/GVL_HW.IoLinkNode2Ch2_Humidity[2] <-> IoLinkNode2_Ch2 (IO-Link Slave)/IO-Link Port2/Port2: process data[4]
//     PlcTask_10ms Inputs/GVL_HW.IoLinkNode2Ch2_Temperature[1] <-> IoLinkNode2_Ch2 (IO-Link Slave)/IO-Link Port2/Port2: process data[0]
//     PlcTask_10ms Inputs/GVL_HW.IoLinkNode2Ch2_Temperature[2] <-> IoLinkNode2_Ch2 (IO-Link Slave)/IO-Link Port2/Port2: process data[1]
//     PlcTask_10ms Inputs/GVL_HW.IoLinkNode2Ch3_Level <-> IoLinkNode2_Ch3 (IO-Link Slave)/IO-Link Port3/Level
//     PlcTask_10ms Inputs/GVL_HW.IoLinkNode2Ch4_DiffPress <-> IoLinkNode2_Ch4 (IO-Link Slave)/IO-Link Port4/Pressure

CONFIGURATION IoT_OPCUA
    RESOURCE PLC ON TwinCAT3
        TASK PlcTask_10ms(INTERVAL := T#10ms, PRIORITY := 20);
        TASK PlcTask_500us(INTERVAL := T#500us, PRIORITY := 23);
        TASK Task_1ms(INTERVAL := T#1ms, PRIORITY := 1);
        PROGRAM PRG_01_MAIN WITH PlcTask_10ms : PRG_01_MAIN;
        PROGRAM Main_500us WITH PlcTask_500us : Main_500us;
        PROGRAM Main_T1ms WITH Task_1ms : Main_T1ms;
    END_RESOURCE
END_CONFIGURATION

// ---- DUTs/AirValveSimSignals.TcDUT
TYPE AirValveSimSignals :
STRUCT 	
	ExtendCmd 		: 	BOOL;
	ExtendFeedback 	: 	BOOL;
	RetractCmd 		: 	BOOL;
	RetractFeedback : 	BOOL;
	SequenceStatus 	: 	INT;
END_STRUCT
END_TYPE

// ---- DUTs/DataModels/DriveState_DataModel.TcDUT
TYPE DriveState_DataModel :
STRUCT
	StartingState 	: STRING(20) := 'Starting';
	RunningState	: STRING(20) := 'Running';
	StoppingState	: STRING(20) := 'Stopping';
	StoppedState	: STRING(20) := 'Stopped';
END_STRUCT
END_TYPE

// ---- DUTs/DataModels/ElectrDevicePeriodicOper_DataModel.TcDUT
(* Electrical device with periodic operation mode *)
TYPE ElectrDevicePeriodicOper_DataModel :
STRUCT
	LineName			: STRING(40);
	MachineName			: STRING(40);
	DeviceName			: STRING(40);
	DeviceState			: STRING(20); // Device state: Running, Stopping, Stopped
	SynchPulse			: BOOL;
	TimeStamp 			: ULINT;
	
	{attribute 'OPC.UA.DA' := '1'}
	{attribute 'OPC.UA.DA.Access' := '1'}			// read only
	{attribute 'OPC.UA.DA.StructuredType' := '1'}
	ElectricalData 		: ElectrDataEthCAT;
END_STRUCT
END_TYPE

// ---- DUTs/DataModels/ElectrDeviceContOper_DataModel.TcDUT
(*Electrical device with continous operation mode*)
TYPE ElectrDeviceContOper_DataModel :
STRUCT
	LineName	: STRING(40);
	MachineName	: STRING(40);
	DeviceName	: STRING(40);
	
	{attribute 'OPC.UA.DA' := '1'}
	{attribute 'OPC.UA.DA.Access' := '1'}			// read only
	{attribute 'OPC.UA.DA.StructuredType' := '1'}
	ElectricalData : ElectrDataModbusTCP;
	
	TimeStamp 	: ULINT;
END_STRUCT
END_TYPE

// ---- DUTs/DataModels/SingleSensor_DataModel.TcDUT
TYPE SingleSensor_DataModel :
STRUCT
	LineName	: STRING(40);
	MachineName	: STRING(40);
	SensorName	: STRING(40);
	SensorValue	: REAL;
	TimeStamp 	: ULINT;
END_STRUCT
END_TYPE

// ---- DUTs/DataModels/SingleState_DataModel.TcDUT
TYPE SingleState_DataModel :
STRUCT
	LineName	: STRING(40);
	MachineName	: STRING(40);
	StateName	: STRING(40);
	StateValue	: INT;
	TimeStamp 	: ULINT;
END_STRUCT
END_TYPE

// ---- DUTs/DataModels/ValveTravelTime_DataModel.TcDUT
TYPE ValveTravelTime_DataModel :
STRUCT

LineName	: STRING(40);
MachineName	: STRING(40);
ValveName	: STRING(40);


{attribute 'DataType' := 'STRING'}
TimeType	: STRING(40);

{attribute 'DataType' := 'INT'}
{attribute 'Unit' := 'ms'}
{attribute 'DisplayName' := 'Time'}
TimeValue 	: INT;

{attribute 'DataType' := 'ULINT'}
TimeStamp : ULINT;

END_STRUCT
END_TYPE

// ---- DUTs/DataModels/VibAccelarationDataModel.TcDUT

TYPE VibAccelarationDataModel :
STRUCT
	LineName			: STRING(40);
	MachineName			: STRING(40);
	SensorName			: STRING(40);
		
	VibAccelTotRmsX		: REAL;
    VibAccelTotRmsY		: REAL;
    VibAccelTotRmsZ		: REAL;

    SensorTemperature	: REAL;
	
	TimeStamp 			: ULINT;	
END_STRUCT
END_TYPE

// ---- DUTs/ElectrDataModbusTCP.TcDUT
TYPE ElectrDataModbusTCP :
STRUCT
	// Power Measurement Data
	// Modbus register from Siemens 7KT PAC1200
	ActPowerPos		:REAL;
	ActPowerNeg		:REAL;
	ReactPowerPos	:REAL;
	ReactPowerNeg	:REAL;
	ApparPowerPos	:REAL;
	ApparPowerNeg	:REAL;
	PowerFact		:REAL;
	LineFreq		:REAL;
	
	//L1 phase data
	ActPowerPosL1	:REAL;
	ActPowerNegL1	:REAL;
	
	ReactPowerPosL1	:REAL;
	ReactPowerNegL1	:REAL;
	
	CurrentL1		:REAL;
	VoltL1			:REAL;
	PowFactL1		:REAL;
	
	//L2 phase data
	ActPowerPosL2	:REAL;
	ActPowerNegL2	:REAL;
	
	ReactPowerPosL2	:REAL;
	ReactPowerNegL2	:REAL;
	
	CurrentL2		:REAL;
	VoltL2			:REAL;
	PowFactL2		:REAL;
	
	//L3 phase data
	ActPowerPosL3	:REAL;
	ActPowerNegL3	:REAL;
	
	ReactPowerPosL3	:REAL;
	ReactPowerNegL3	:REAL;
	
	CurrentL3		:REAL;
	VoltL3			:REAL;
	PowFactL3		:REAL;
END_STRUCT
END_TYPE

// ---- DUTs/ElectrDataEthCAT.TcDUT
TYPE ElectrDataEthCAT :
STRUCT
	//Power Measurement Data
	// ************* total measurements ***********
	ActPowerTot		:REAL;
	ReactPowerTot	:REAL;
	ApparPowerTot	:REAL;
	PowerFact		:REAL;
	PQF				:REAL;	// power quality factor
	
	//************* L1 phase data *****************
	ActPowerL1		:REAL;
	ReactPowerL1	:REAL;
	ApparPowerL1	:REAL;
	
	CurrentL1		:REAL;
	VoltL1			:REAL;
	PowFactL1		:REAL;
	VoltL1_THD		:REAL;	// THD of voltage
	//VoltL1_harm		:ARRAY [0..41] OF REAL;		// [% of fundamental rms] 0 => DC component, 1 => fundamental wave, 2=> 2nd harmonic, 3=> 3rd harmonic
	
	CurrentL1_THD	:REAL;	// THD of current
	CurrentL1_Harm	:ARRAY [0..41] OF REAL;		// [% of fundamental rms] 0 => DC component, 1 => fundamental wave, 2=> 2nd harmonic, 3=> 3rd harmonic
	
	//************* L2 phase data *****************
	ActPowerL2		:REAL;
	ReactPowerL2	:REAL;
	ApparPowerL2	:REAL;
	
	CurrentL2		:REAL;
	VoltL2			:REAL;
	PowFactL2		:REAL;
	VoltL2_THD		:REAL;	// THD of voltage
	//VoltL2_harm		:ARRAY [0..41] OF REAL;		// [% of fundamental rms] 0 => DC component, 1 => fundamental wave, 2=> 2nd harmonic, 3=> 3rd harmonic
	
	CurrentL2_THD	:REAL;	// THD of current
	CurrentL2_Harm	:ARRAY [0..41] OF REAL;		// [% of fundamental rms] 0 => DC component, 1 => fundamental wave, 2=> 2nd harmonic, 3=> 3rd harmonic
	
	
	//************* L3 phase data *****************
	
	ActPowerL3		:REAL;
	ReactPowerL3	:REAL;
	ApparPowerL3	:REAL;
	
	CurrentL3		:REAL;
	VoltL3			:REAL;
	PowFactL3		:REAL;
	VoltL3_THD		:REAL;	// THD of voltage
	//VoltL3_harm		:ARRAY [0..41] OF REAL;		// [% of fundamental rms] 0 => DC component, 1 => fundamental wave, 2=> 2nd harmonic, 3=> 3rd harmonic
	
	CurrentL3_THD	:REAL;	// THD of current
	CurrentL3_Harm	:ARRAY [0..41] OF REAL;		// [% of fundamental rms] 0 => DC component, 1 => fundamental wave, 2=> 2nd harmonic, 3=> 3rd harmonic

END_STRUCT
END_TYPE

// ---- POUs/EL3443/EL3443/DUTs/E_EL3443_Phase.TcDUT
(*This enum is equivalent to the selectors from the documentation " Confirmation of variable output values 1 - 4"*)
{attribute 'qualified_only'}
TYPE E_EL3443_Phase :
(
    nPhaseL1_OFFSET := 256,     //Offset Channel 1(Phase L1). The offset is added to the base selector     
    nPhaseL2_OFFSET := 512,     //Offset Channel 2(Phase L2). The offset is added to the base selector
    nPhaseL3_OFFSET := 768,     //Offset Channel 3(Phase L3). The offset is added to the base selector
    
    U_RMS := 1,					// [V] (Real Selector: 1 (Examp.: 257 = 1 + 256 for ch. 1)) RMS value of the voltage
    U_peak := 2,                // [V] (Real Selector: 2 (Examp.: 770 = 2 + 768 for ch. 3)) Peak value of the instantaneous voltage in the last interval
    U_Last_Zero_Cross := 3,     // [V] (UINT Selector: 3) DC time of the penultimate voltage zero crossing
    U_RMS_Minimum := 4,         // [V] (Real Selector: 4) Minimum RMS value of the voltage in the last interval
    U_RMS_Maximum := 5,         // [V] (Real Selector: 5) Maximum RMS value of the voltage in the last interval
    ULL := 6,                   // [V] (Real Selector: 6) RMS value of the phase-to-phase voltage (Channel 1: U_L1L2; Channel 1: U_L2L3; Channel 3: U_L3L1) 
    I_RMS := 8,                 // [A] (Real Selector: 8) RMS value of the current
    I_peak := 9,                // [A] (Real Selector: 9) Peak value of the instantaneous current in the last interval
    I_RMS_Minimum := 11,        // [A] (Real Selector: 11) Minimum RMS value of the current in the last interval
    I_RMS_Maximum := 12,        // [A] (Real Selector: 12) Maximum RMS value of the current in the last interval
    Frequency := 17,            // [Hz] (Real Selector: 17) Frequency of this phase
    Phi := 21,                  // [°] (Real Selector: 21) Phase angle of the fundamental wave
    Cos_phi := 22,              // [-] (Real Selector: 22) Cosine of the fundamental wave phase angle
    Power_Factor := 23,         // [-] (Real Selector: 23) Power factor
    P := 26,                    // [W] (Real Selector: 26) Active power
    Pavg := 27,                 // [W] (Real Selector: 27) Average active power during the last interval
    Pmin := 28,                 // [W] (Real Selector: 28) Minimum active power in the last interval
    Pmax := 29,                 // [W] (Real Selector: 29) Maximum active power in the last interval
    S_ := 32,                   // [VA] (Real Selector: 32) Apparent power
    Savg := 33,                 // [VA] (Real Selector: 33) Average apparent power during the last interval
    Smin := 34,                 // [VA] (Real Selector: 34) Minimum apparent power in last interval
    Smax := 35,                 // [VA] (Real Selector: 35) Minimum apparent power in last interval
    Q := 38,                    // [Var] (Real Selector: 38) Reactive power
    Qavg := 39,                 // [Var] (Real Selector: 39) Average reactive power average during the last interval
    Qmin := 40,                 // [Var] (Real Selector: 40) Minimum reactive power in the last interval
    Qmax := 41,                 // [Var] (Real Selector: 41) Maximum reactive power in the last interval
    EP := 45,                   // [mhW] (UINT Selector: 45) Recorded active energy
    EP_pos := 46,               // [mhW] (UINT Selector: 46) Received active energy
    EP_neg := 47,               // [mhW] (UINT Selector: 47) Supplied active energy
	EP_interval:= 48, 			// [mhW] (UINT Selector: 48) Recorded active energy in the last interval
	EP_pos_interval:= 49, 		// [mhW] (UINT Selector: 49) Received active energy in the last interval
	EP_neg_interval:= 50, 		// [mhW] (UINT Selector: 50) Supplied active energy in the last interval
    ES := 51,                   // [mhW] (UINT Selector: 51) Apparent energy
    ES_pos := 52,               // [mhW] (UINT Selector: 52) Apparent energy
    ES_neg := 53,               // [mhW] (UINT Selector: 53) Apparent energy
	ES_interval:= 54, 			// [mhW] (UINT Selector: 54) Apparent energy in the last interval
	ES_pos_interval:= 55, 		// [mhW] (UINT Selector: 55) Apparent energy in the last interval
	ES_neg_interval:= 56, 		// [mhW] (UINT Selector: 56) Apparent energy in the last interval
    EQ_ := 57,                  // [mhW] (UINT Selector: 57) Reactive energy
    EQ_pos := 58,               // [mhW] (UINT Selector: 58) Reactive energy
    EQ_neg := 59,               // [mhW] (UINT Selector: 59) Reactive energy
	EQ_interval:= 60, 			// [mhW] (UINT Selector: 60) Reactive energy in the last interval
	EQ_pos_interval:= 61, 		// [mhW] (UINT Selector: 62) Reactive energy in the last interval
	EQ_neg_interval:= 62, 		// [mhW] (UINT Selector: 63) Reactive energy in the last interval
    THD_U := 95,                // [-] (Real Selector: 95) "Total Harmonic Distortion" is the distortion factor of the voltage. It indicates the ratio of the harmonic components of an oscillation relative to its fundamental.
    RMS_fund_U := 98,           // [V] (Real Selector: 98) Amplitude of the fundamental wave
    F_Ref_U := 99,              // [Hz] (Real Selector: 99) Reference frequency of the voltage harmonic: Specifies the underlying fundamental frequency, e.g.: 50 or 60 Hz.
    Harmonics_U := 100,         // [% of the fundamental wave] (Real Selector: 100-141) 0 => DC component, 1 => fundamental wave, 2=> 2nd harmonic, 3=> 3rd harmonic
    THD_I := 165,               // [-] (Real Selector: 165) "Total Harmonic Distortion" is the distortion factor of the current. It indicates the ratio of the harmonic components of an oscillation relative to its fundamental.
    TDD_I := 166,               // [% of the maximum current] (Real Selector: 166) "Total Demand Distortion" indicates the ratio between the current harmonics and the maximum current (EL3443: 1A and EL3443-0010: 5A)
    RMS_fund_I := 168,          // [A] (Real Selector: 168) Amplitude of the fundamental wave
    F_Ref_I := 169,             // [Hz] (Real Selector: 169) Reference frequency of the current harmonic: Specifies the underlying fundamental frequency, e.g.: 50 or 60 Hz.
    Harmonics_I := 170,         // [% of the fundamental wave] (Real Selector: 170-211) 0 => DC component, 1 => fundamental wave, 2=> 2nd harmonic, 3=> 3rd harmonic
    Error_INDEX_Not_Valid := 255 // [-] (Real Selector: 255) Error message: The selected index is not available.
)UINT;
END_TYPE

// ---- POUs/EL3443/EL3443/DUTs/E_EL3443_Total.TcDUT
(*This enum is equivalent to the selectors from the documentation " Confirmation of variable output values 1 - 4"*)
{attribute 'qualified_only'}
TYPE E_EL3443_Total :
(
    nTotal_OFFSET := 1024,           // Offset for total values. The offset is added to the base selector
    
    In_RMS := 8,                     // [A]  (Real Selector: 1032 (= 1024 + 8))  Calculated RMS value of the neutral current
    Power_Factor := 23,              // [-]  (Real Selector: 1047 (= 1024 + 23))  Total power factor over all phases
    Ptot := 26,                      // [W]  (Real Selector: 1050 (= 1024 + 26))  Total active power
    Ptotavg := 27,                   // [W]  (Real Selector: 1051 (= 1024 + 27))  Average total active power during the last interval
    Ptotmin := 28,                   // [W]  (Real Selector: 1052 (= 1024 + 28))  Minimum total active power in the last interval
    Ptotmax := 29,                   // [W]  (Real Selector: 1053 (= 1024 + 29))  Maximum total active power in the last interval
    Stot := 32,                      // [VA]  (Real Selector: 1056 (= 1024 + 32))  Total apparent power
    Stotavg := 33,                   // [VA]  (Real Selector: 1057 (= 1024 + 33))  Average total apparent power during the last interval
    Stotmin := 34,                   // [VA]  (Real Selector: 1058 (= 1024 + 34))  Minimum total apparent power in the last interval
    Stotmax := 35,                   // [VA]  (Real Selector: 1059 (= 1024 + 35))  Maximum total apparent power in the last interval
    Qtot := 38,                      // [Var]  (Real Selector: 1062 (= 1024 + 38))  Total reactive power
    Qtotavg := 39,                   // [Var]  (Real Selector: 1063 (= 1024 + 39))  Average total reactive power during the last interval
    Qtotmin := 40,                   // [Var]  (Real Selector: 1064 (= 1024 + 40))  Minimum total reactive power in the last interval
    Qtotmax := 41,                   // [Var]  (Real Selector: 1065 (= 1024 + 41))  Maximum total reactive power in the last interval
    Eptot := 45,                     // [mWh]  (ULINT Selector: 1069 (= 1024 + 45))  Balanced total active energy
    EPtot_pos := 46,                 // [mWh]  (ULINT Selector: 1070 (= 1024 + 46))  Related total active energy
    EPtot_neg := 47,                 // [mWh]  (ULINT Selector: 1071 (= 1024 + 47))  Input total active energy
    Eptot_interval := 48,           // [mWh]  (ULINT Selector: 1072 (= 1024 + 48))  Balanced total active energy in last interval
    EPtot_pos_interval := 49,       // [mWh]  (ULINT Selector: 1073 (= 1024 + 49))  Total active energy related in the last interval
    EPtot_neg_interval := 50,       // [mWh]  (ULINT Selector: 1074 (= 1024 + 50))  Input total active energy the last interval
    EStot := 51,                     // [mWh]  (ULINT Selector: 1075 (= 1024 + 51))  Total apparent energy
    EStot_pos := 52,                 // [mWh]  (ULINT Selector: 1076 (= 1024 + 52))  Total apparent energy
    EStot_neg := 53,                 // [mWh]  (ULINT Selector: 1077 (= 1024 + 53))  Total apparent energy
    EStot_interval := 54,           // [mWh]  (ULINT Selector: 1078 (= 1024 + 54))  Total apparent energy in the last interval
    EStot_pos_interval := 55,       // [mWh]  (ULINT Selector: 1079 (= 1024 + 55))  Total apparent energy in the last interval
    EStot_neg_interval := 56,       // [mWh]  (ULINT Selector: 1080 (= 1024 + 56))  Total apparent energy in the last interval
    EQtot := 57,                     // [mWh]  (ULINT Selector: 1081 (= 1024 + 57))  Total reactive energy
    EQtot_pos := 58,                 // [mWh]  (ULINT Selector: 1082 (= 1024 + 58))  Total reactive energy
    EQtot_neg := 59,                 // [mWh]  (ULINT Selector: 1083 (= 1024 + 59))  Total reactive energy
    EQtot_interval := 60,           // [mWh]  (ULINT Selector: 1084 (= 1024 + 60))  Total reactive energy in the last interval
    EQtot_pos_interval := 61,       // [mWh]  (ULINT Selector: 1085 (= 1024 + 61))  Total reactive energy in the last interval
    EQtot_neg_interval := 62,       // [mWh]  (ULINT Selector: 1086 (= 1024 + 62))  Total reactive energy in the last interval
    PhiL1L2 := 70,                   // [°]  (Real Selector: 1094 (= 1024 + 70))  Phase shift angle between phase L1 and L2
    PhiL1L3 := 71,                   // [°]  (Real Selector: 1095 (= 1024 + 71))  Phase shift angle between phase L1 and L3
    Unbalance := 72,                 // [-]  (Real Selector: 1096 (= 1024 + 72))  Ratio between negative and positive voltage system
    PQF := 80,                       // [-]  (Real Selector: 1104 (= 1024 + 80))  Power quality factor
    PQF_Avg := 81,                   // [-]  (Real Selector: 1105 (= 1024 + 81))  Average value of the power quality factor during the last interval
    PQF_MIN := 82,                   // [-]  (Real Selector: 1106 (= 1024 + 82))  Minimum power quality factor in the last interval
    PQF_MAX := 83                    // [-]  (Real Selector: 1107 (= 1024 + 83))  Maximum power quality factor in the last interval
)UINT;      
END_TYPE

// ---- POUs/EL3443/EL3443/DUTs/ST_EL3443_MUX_REAL.TcDUT
TYPE ST_EL3443_MUX_REAL :
STRUCT
    nSelector : UINT := E_EL3443_Phase.Error_INDEX_Not_Valid;
    fValueRef : REFERENCE TO REAL;
END_STRUCT
END_TYPE

// ---- POUs/EL3443/EL3443/DUTs/ST_EL3443_MUX_ULINT.TcDUT
TYPE ST_EL3443_MUX_ULINT :
STRUCT
    nSelector : UINT := E_EL3443_Phase.Error_INDEX_Not_Valid;
    nValueRef : POINTER TO ULINT;
END_STRUCT
END_TYPE

// ---- POUs/EL3443/EL3443/DUTs/ST_EL3443_StatusLx.TcDUT
TYPE ST_EL3443_StatusLx :
STRUCT
    bStatus_Voltage_Sign_Bit : BOOL;             //Voltage Sign Bit - Indicates the sign of the current sine wave voltage: 1 = U > 0V, 0 = U < 0V
    bStatus_Overvoltage : BOOL;                  //Overvoltage - Maximum measurable voltage is exceeded.
    bStatus_Overcurrent : BOOL;                  //Overcurrent - Maximum measurable current is exceeded.
    bStatus_Inaccurate_Voltage : BOOL;           //Inaccurate Voltage - The measured voltage value is smaller than the value entered in CoE object "F800:15 Inaccurate Threshold Voltage".
    bStatus_Inaccurate_Current : BOOL;           //Inaccurate Current - The measured current value is smaller than the value entered in CoE object "F800:16 Inaccurate Threshold Current".
    bStatus_Voltage_Guard_Warning : BOOL;        //Voltage Guard Warning - A warning limit of the voltage monitor has been breached.
    bStatus_Voltage_Guard_Error : BOOL;          //Voltage Guard Error - An error limit of the voltage monitor has been breached.
    bStatus_Current_Guard_Warning : BOOL;        //Voltage Current Warning - A warning limit of the Current monitor has been breached.
    bStatus_Current_Guard_Error : BOOL;          //Voltage Current Error - An error limit of the Current monitor has been breached.
    bStatus_TxPDO_Toggle : BOOL;                 //TxPDO Toggle - The TxPDO toggle is toggled by the slave when the data of the associated TxPDO is updated.
    fBasic_Voltage : REAL;                       //Voltage - RMS value of the voltage in V
    fBasic_Current : REAL;                       //Current - RMS value of the current in A
    fPower_Active_Power : REAL;                  //Active power Active power in W
    fPower_Apparent_Power : REAL;                //Apparent Power Apparent power in VA
    fPower_Reactive_Power : REAL;                //Reactive Power Reactive power in var
    fPower_Power_Factor : REAL;                  //Power Factor Power factor
    nTiming_Voltage_Last_Zero_Crossing : ULINT;  //Voltage Last Zero Crossing - Last detected voltage zero crossing as distributed clock time
END_STRUCT
END_TYPE

// ---- POUs/EL3443/EL3443/DUTs/ST_EL3443_StatusTotal.TcDUT
TYPE ST_EL3443_StatusTotal :
STRUCT
    bStatus_System_State : BOOL;                        //System State - Overall system state (as a logical disjunction of voltage guard errors, phase sequence, overvoltage, overcurrent and frequency guard errors)
    bStatus_Grid_Direction : BOOL;                      //Grid Direction - Phase sequence L1 - L2 - L3 correctly detected (with clockwise 3-phase mains)
    bStatus_Frequency_Guard_Warning : BOOL;             //Frequency Guard Warning - A warning limit of the frequency monitor has been breached.
    bStatus_Frequency_Guard_Error : BOOL;               //Frequency Guard Error - An error limit of the frequency monitor has been breached.
    bStatus_Neutral_Current_Guard_Warning : BOOL;       //Neutral Current Guard Warning - A warning limit of the neutral conductor current monitor has been breached.
    bStatus_Neutral_Current_Guard_Error : BOOL;         //Neutral Current Guard Error - An error limit of the neutral conductor current monitor has been breached.
    bStatus_Active_Power_Guard_Warning : BOOL;          //Active Power Guard Warning - A warning limit of the active power monitor has been breached.
    bStatus_Active_Power_Guard_Error : BOOL;            //Active Power Guard Error - An error limit of the active power monitor has been breached.
    bStatus_Apparent_Power_Guard_Warning : BOOL;        //Apparent Power Guard Warning - A warning limit of the apparent power monitor has been breached.
    bStatus_Apparent_Power_Guard_Error : BOOL;          //Apparent Power Guard Error - An error limit of the apparent power monitor has been breached.
    bStatus_Power_Quality_Guard_Warning : BOOL;         //Power Quality Guard Warning - A warning limit of the PQF monitor has been breached.
    bStatus_Power_Quality_Guard_Error : BOOL;           //Power Quality Guard Error - An error limit of the PQF monitor has been breached.
    bStatus_TxPDO_State : BOOL;                         //TxPDO State - TRUE for general error
    bStatus_TxPDO_Toggle : BOOL;                        //TxPDO Toggle - The TxPDO toggle is toggled by the slave when the data of the associated TxPDO is updated.
    fStatus_Power_Quality_Factor : REAL;                //Power Quality Factor - Analog value of the voltage quality between 1.0 and 0 (see basic function principles - Power Quality Factor)
    fBasic_Frequency : REAL;                            //Frequency - Frequency in Hz
    fBasic_Power_Factor : REAL;                         //Power Factor - Power factor
    fBasic_Calculated_Neutral_Line_Current : REAL; 		//Calculated Neutral Line Current - Calculated RMS value of the neutral conductor current in A
END_STRUCT                                              
END_TYPE

// ---- POUs/EL3443/EL3443/DUTs/ST_EL3443_VariantLx.TcDUT
TYPE ST_EL3443_VariantLx :
STRUCT
    fU_RMS : REAL;						// [V] (Real Selector: 1 (Examp.: 257 = 1 + 256 for ch. 1)) RMS value of the voltage
    fU_peak : REAL;						// [V] (Real Selector: 2 (Examp.: 770 = 2 + 768 for ch. 3)) Peak value of the instantaneous voltage in the last interval
    nU_Last_Zero_Cross : ULINT;			// [V] (UINT Selector: 3) DC time of the penultimate voltage zero crossing
    fU_RMS_Minimum : REAL;				// [V] (Real Selector: 4) Minimum RMS value of the voltage in the last interval
    fU_RMS_Maximum : REAL;				// [V] (Real Selector: 5) Maximum RMS value of the voltage in the last interval
    fULL : REAL;						// [V] (Real Selector: 6) RMS value of the phase-to-phase voltage (Channel 1: U_L1L2; Channel 1: U_L2L3; Channel 3: U_L3L1) 
    fI_RMS : REAL;						// [A] (Real Selector: 8) RMS value of the current
    fI_peak : REAL;						// [A] (Real Selector: 9) Peak value of the instantaneous current in the last interval
    fI_RMS_Minimum : REAL;				// [A] (Real Selector: 11) Minimum RMS value of the current in the last interval
    fI_RMS_Maximum : REAL;				// [A] (Real Selector: 12) Maximum RMS value of the current in the last interval
    fFrequency : REAL;					// [Hz] (Real Selector: 17) Frequency of this phase
    fPhi : REAL;						// [°] (Real Selector: 21) Phase angle of the fundamental wave
    fCOS_phi : REAL;					// [-] (Real Selector: 22) Cosine of the fundamental wave phase angle
    fPower_Factor : REAL;				// [-] (Real Selector: 23) Power factor
    fP : REAL;							// [W] (Real Selector: 26) Active power
    fPavg : REAL;						// [W] (Real Selector: 27) Average active power during the last interval
    fPmin : REAL;						// [W] (Real Selector: 28) Minimum active power in the last interval
    fPmax : REAL;						// [W] (Real Selector: 29) Maximum active power in the last interval
    fS : REAL;							// [VA] (Real Selector: 32) Apparent power
    fSavg : REAL;						// [VA] (Real Selector: 33) Average apparent power during the last interval
    fSmin : REAL;						// [VA] (Real Selector: 34) Minimum apparent power in last interval
    fSmax : REAL;						// [VA] (Real Selector: 35) Minimum apparent power in last interval
    fQ : REAL;							// [Var] (Real Selector: 38) Reactive power
    fQavg : REAL;						// [Var] (Real Selector: 39) Average reactive power average during the last interval
    fQmin : REAL;						// [Var] (Real Selector: 40) Minimum reactive power in the last interval
    fQmax : REAL;						// [Var] (Real Selector: 41) Maximum reactive power in the last interval
    nEP : LINT;							// [mhW] (LINT Selector: 45) Recorded active energy
    nEP_pos : ULINT;					// [mhW] (UINT Selector: 46) Received active energy
    nEP_neg : ULINT;					// [mhW] (UINT Selector: 47) Supplied active energy
	nEP_interval : LINT;				// [mhW] (LINT Selector: 48) Recorded active energy in the last interval
	nEP_pos_interval : ULINT;			// [mhW] (UINT Selector: 49) Received active energy in the last interval
	nEP_neg_interval : ULINT;			// [mhW] (UINT Selector: 50) Supplied active energy in the last interval
    nES : LINT;							// [mhW] (LINT Selector: 51) Apparent energy
    nES_pos : ULINT;					// [mhW] (UINT Selector: 52) Apparent energy
    nES_neg : ULINT;					// [mhW] (UINT Selector: 53) Apparent energy
	nES_interval : LINT;				// [mhW] (LINT Selector: 54) Apparent energy in the last interval
	nES_pos_interval : ULINT;			// [mhW] (UINT Selector: 55) Apparent energy in the last interval
	nES_neg_interval : ULINT;			// [mhW] (UINT Selector: 56) Apparent energy in the last interval
    nEQ : LINT;							// [mhW] (LINT Selector: 57) Reactive energy
    nEQ_pos : ULINT;					// [mhW] (UINT Selector: 58) Reactive energy
    nEQ_neg : ULINT;					// [mhW] (UINT Selector: 59) Reactive energy
	nEQ_interval : LINT;				// [mhW] (LINT Selector: 60) Reactive energy in the last interval
	nEQ_pos_interval : ULINT;			// [mhW] (UINT Selector: 62) Reactive energy in the last interval
	nEQ_neg_interval : ULINT;			// [mhW] (UINT Selector: 63) Reactive energy in the last interval
    fTHD_U : REAL;						// [-] (Real Selector: 95) "Total Harmonic Distortion" is the distortion factor of the voltage. It indicates the ratio of the harmonic components of an oscillation relative to its fundamental.
    fRMS_fund_U : REAL;					// [V] (Real Selector: 98) Amplitude of the fundamental wave
    fF_Ref_U : REAL;					// [Hz] (Real Selector: 99) Reference frequency of the voltage harmonic: Specifies the underlying fundamental frequency, e.g.: 50 or 60 Hz.
    fHarmonics_U : ARRAY [0..41] OF REAL;// [% of the fundamental wave] (Real Selector: 100-141) 0 => DC component, 1 => fundamental wave, 2=> 2nd harmonic, 3=> 3rd harmonic
    fTHD_I : REAL;						// [-] (Real Selector: 165) "Total Harmonic Distortion" is the distortion factor of the current. It indicates the ratio of the harmonic components of an oscillation relative to its fundamental.
    fTDD_I : REAL;						// [% of the maximum current] (Real Selector: 166) "Total Demand Distortion" indicates the ratio between the current harmonics and the maximum current (EL3443: 1A and EL3443-0010: 5A)
    fRMS_fund_I : REAL;					// [A] (Real Selector: 168) Amplitude of the fundamental wave
    fF_Ref_I : REAL;					// [Hz] (Real Selector: 169) Reference frequency of the current harmonic: Specifies the underlying fundamental frequency, e.g.: 50 or 60 Hz.
    fHarmonics_I : ARRAY [0..41] OF REAL;// [% of the fundamental wave] (Real Selector: 170-211) 0 => DC component, 1 => fundamental wave, 2=> 2nd harmonic, 3=> 3rd harmonic
END_STRUCT
END_TYPE

// ---- POUs/EL3443/EL3443/DUTs/ST_EL3443_VariantTotal.TcDUT
TYPE ST_EL3443_VariantTotal :
STRUCT
    fIn_RMS : REAL; 			// [A]  (Real Selector: 1032 (= 1024 + 8))  Calculated RMS value of the neutral current
    fPower_Factor : REAL; 		// [-]  (Real Selector: 1047 (= 1024 + 23))  Total power factor over all phases
    fPtot : REAL; 				// [W]  (Real Selector: 1050 (= 1024 + 26))  Total active power
    fPtotavg : REAL; 			// [W]  (Real Selector: 1051 (= 1024 + 27))  Average total active power during the last interval
    fPtotmin : REAL; 			// [W]  (Real Selector: 1052 (= 1024 + 28))  Minimum total active power in the last interval
    fPtotmax : REAL; 			// [W]  (Real Selector: 1053 (= 1024 + 29))  Maximum total active power in the last interval
    fStot : REAL; 				// [VA]  (Real Selector: 1056 (= 1024 + 32))  Total apparent power
    fStotavg : REAL; 			// [VA]  (Real Selector: 1057 (= 1024 + 33))  Average total apparent power during the last interval
    fStotmin : REAL; 			// [VA]  (Real Selector: 1058 (= 1024 + 34))  Minimum total apparent power in the last interval
    fStotmax : REAL; 			// [VA]  (Real Selector: 1059 (= 1024 + 35))  Maximum total apparent power in the last interval
    fQtot : REAL; 				// [Var]  (Real Selector: 1062 (= 1024 + 38))  Total reactive power
    fQtotavg : REAL; 			// [Var]  (Real Selector: 1063 (= 1024 + 39))  Average total reactive power during the last interval
    fQtotmin : REAL; 			// [Var]  (Real Selector: 1064 (= 1024 + 40))  Minimum total reactive power in the last interval
    fQtotmax : REAL; 			// [Var]  (Real Selector: 1065 (= 1024 + 41))  Maximum total reactive power in the last interval
    nEptot : LINT; 				// [mWh]  (LINT Selector: 1069 (= 1024 + 45))  Balanced total active energy
    nEPtot_pos : ULINT; 		// [mWh]  (ULINT Selector: 1070 (= 1024 + 46))  Related total active energy
    nEPtot_neg : ULINT; 		// [mWh]  (ULINT Selector: 1071 (= 1024 + 47))  Input total active energy
    nEptot_interval : LINT; 	// [mWh]  (LINT Selector: 1072 (= 1024 + 48))  Balanced total active energy in last interval
    nEPtot_pos_interval : ULINT;// [mWh]  (ULINT Selector: 1073 (= 1024 + 49))  Total active energy related in the last interval
    nEPtot_neg_interval : ULINT;// [mWh]  (ULINT Selector: 1074 (= 1024 + 50))  Input total active energy the last interval
    nEStot : LINT; 				// [mWh]  (LINT Selector: 1075 (= 1024 + 51))  Total apparent energy
    nEStot_pos : ULINT; 		// [mWh]  (ULINT Selector: 1076 (= 1024 + 52))  Total apparent energy
    nEStot_neg : ULINT; 		// [mWh]  (ULINT Selector: 1077 (= 1024 + 53))  Total apparent energy
    nEStot_interval : LINT; 	// [mWh]  (LINT Selector: 1078 (= 1024 + 54))  Total apparent energy in the last interval
    nEStot_pos_interval : ULINT;// [mWh]  (ULINT Selector: 1079 (= 1024 + 55))  Total apparent energy in the last interval
    nEStot_neg_interval : ULINT;// [mWh]  (ULINT Selector: 1080 (= 1024 + 56))  Total apparent energy in the last interval
    nEQtot : LINT; 				// [mWh]  (LINT Selector: 1081 (= 1024 + 57))  Total reactive energy
    nEQtot_pos : ULINT; 		// [mWh]  (ULINT Selector: 1082 (= 1024 + 58))  Total reactive energy
    nEQtot_neg : ULINT; 		// [mWh]  (ULINT Selector: 1083 (= 1024 + 59))  Total reactive energy
    nEQtot_interval : LINT; 	// [mWh]  (LINT Selector: 1084 (= 1024 + 60))  Total reactive energy in the last interval
    nEQtot_pos_interval : ULINT;// [mWh]  (ULINT Selector: 1085 (= 1024 + 61))  Total reactive energy in the last interval
    nEQtot_neg_interval : ULINT;// [mWh]  (ULINT Selector: 1086 (= 1024 + 62))  Total reactive energy in the last interval
    fPhiL1L2 : REAL; 			// [°]  (Real Selector: 1094 (= 1024 + 70))  Phase shift angle between phase L1 and L2
    fPhiL1L3 : REAL; 			// [°]  (Real Selector: 1095 (= 1024 + 71))  Phase shift angle between phase L1 and L3
    fUnbalance : REAL; 			// [-]  (Real Selector: 1096 (= 1024 + 72))  Ratio between negative and positive voltage system
    fPQF : REAL; 				// [-]  (Real Selector: 1104 (= 1024 + 80))  Power quality factor
    fPQF_Avg : REAL; 			// [-]  (Real Selector: 1105 (= 1024 + 81))  Average value of the power quality factor during the last interval
    fPQF_Min : REAL; 			// [-]  (Real Selector: 1106 (= 1024 + 82))  Minimum power quality factor in the last interval
    fPQF_Max : REAL; 			// [-]  (Real Selector: 1107 (= 1024 + 83))  Maximum power quality factor in the last interval
END_STRUCT
END_TYPE

// ---- POUs/EL3443/EL3443/DUTs/ST_EL3443_VariantValues.TcDUT
{attribute 'no-analysis'}
TYPE ST_EL3443_VariantValues :
STRUCT
	astLx 			: ARRAY[1..3] OF ST_EL3443_VariantLx;
	stTotal 		: ST_EL3443_VariantTotal;
END_STRUCT
END_TYPE

// ---- POUs/EL3443/EL3443_DPM/DUTs/E_EL3443_DPM_Phase.TcDUT
(*This enum is equivalent to the selectors from the documentation " Confirmation of variable output values 1 - 4"*)
{attribute 'qualified_only'}
TYPE E_EL3443_DPM_Phase :
(
    nPhaseL1_OFFSET := 256,      //Offset Channel 1(Phase L1). The offset is added to the base selector     
    nPhaseL2_OFFSET := 512,      //Offset Channel 2(Phase L2). The offset is added to the base selector
    nPhaseL3_OFFSET := 768,      //Offset Channel 3(Phase L3). The offset is added to the base selector
    
    U_RMS := 1,                  // [V] (Real Selector: 1 (Examp.: 257 = 1 + 256 for ch. 1)) RMS value of the voltage
    U_peak := 2,                 // [V] (Real Selector: 2 (Examp.: 770 = 2 + 768 for ch. 3)) Peak value of the instantaneous voltage in the last interval
    U_Last_Zero_Cross := 3,      // [V] (UINT Selector: 3) DC time of the penultimate voltage zero crossing
    U_RMS_Minimum := 4,          // [V] (Real Selector: 4) Minimum RMS value of the voltage in the last interval
    U_RMS_Maximum := 5,          // [V] (Real Selector: 5) Maximum RMS value of the voltage in the last interval
    ULL := 6,                    // [V] (Real Selector: 6) RMS value of the phase-to-phase voltage (Channel 1: U_L1L2; Channel 1: U_L2L3; Channel 3: U_L3L1) 
    I_RMS := 8,                  // [A] (Real Selector: 8) RMS value of the current
    I_peak := 9,                 // [A] (Real Selector: 9) Peak value of the instantaneous current in the last interval
    I_RMS_Minimum := 11,         // [A] (Real Selector: 11) Minimum RMS value of the current in the last interval
    I_RMS_Maximum := 12,         // [A] (Real Selector: 12) Maximum RMS value of the current in the last interval
    Frequency := 17,             // [Hz] (Real Selector: 17) Frequency of this phase
    Phi := 21,                   // [°] (Real Selector: 21) Phase angle of the fundamental wave
    Cos_phi := 22,               // [-] (Real Selector: 22) Cosine of the fundamental wave phase angle
    Power_Factor := 23,          // [-] (Real Selector: 23) Power factor
    P := 26,                     // [W] (Real Selector: 26) Active power
    Pavg := 27,                  // [W] (Real Selector: 27) Average active power during the last interval
    Pmin := 28,                  // [W] (Real Selector: 28) Minimum active power in the last interval
    Pmax := 29,                  // [W] (Real Selector: 29) Maximum active power in the last interval
    S_ := 32,                    // [VA] (Real Selector: 32) Apparent power
    Savg := 33,                  // [VA] (Real Selector: 33) Average apparent power during the last interval
    Smin := 34,                  // [VA] (Real Selector: 34) Minimum apparent power in last interval
    Smax := 35,                  // [VA] (Real Selector: 35) Minimum apparent power in last interval
    Q := 38,                     // [Var] (Real Selector: 38) Reactive power
    Qavg := 39,                  // [Var] (Real Selector: 39) Average reactive power average during the last interval
    Qmin := 40,                  // [Var] (Real Selector: 40) Minimum reactive power in the last interval
    Qmax := 41,                  // [Var] (Real Selector: 41) Maximum reactive power in the last interval
    EP := 45,                    // [mhW] (UINT Selector: 45) Recorded active energy
    EP_pos := 46,                // [mhW] (UINT Selector: 46) Received active energy
    EP_neg := 47,                // [mhW] (UINT Selector: 47) Supplied active energy
	EP_interval := 48, 			// [mhW] (UINT Selector: 48) Recorded active energy in the last interval
	EP_pos_interval := 49, 		// [mhW] (UINT Selector: 49) Received active energy in the last interval
	EP_neg_interval := 50, 		// [mhW] (UINT Selector: 50) Supplied active energy in the last interval
    ES := 51,                    // [mhW] (UINT Selector: 51) Apparent energy
    ES_pos := 52,                // [mhW] (UINT Selector: 52) Apparent energy
    ES_neg := 53,                // [mhW] (UINT Selector: 53) Apparent energy
	ES_interval := 54, 			// [mhW] (UINT Selector: 54) Apparent energy in the last interval
	ES_pos_interval := 55, 		// [mhW] (UINT Selector: 55) Apparent energy in the last interval
	ES_neg_interval := 56, 		// [mhW] (UINT Selector: 56) Apparent energy in the last interval
    EQ_ := 57,                   // [mhW] (UINT Selector: 57) Reactive energy
    EQ_pos := 58,                // [mhW] (UINT Selector: 58) Reactive energy
    EQ_neg := 59,                // [mhW] (UINT Selector: 59) Reactive energy
	EQ_interval := 60, 			// [mhW] (UINT Selector: 60) Reactive energy in the last interval
	EQ_pos_interval := 61, 		// [mhW] (UINT Selector: 62) Reactive energy in the last interval
	EQ_neg_interval := 62, 		// [mhW] (UINT Selector: 63) Reactive energy in the last interval
    THD_U := 95,                 // [-] (Real Selector: 95) "Total Harmonic Distortion" is the distortion factor of the voltage. It indicates the ratio of the harmonic components of an oscillation relative to its fundamental.
    RMS_fund_U := 98,            // [V] (Real Selector: 98) Amplitude of the fundamental wave
    F_Ref_U := 99,               // [Hz] (Real Selector: 99) Reference frequency of the voltage harmonic: Specifies the underlying fundamental frequency, e.g.: 50 or 60 Hz.
    Harmonics_U := 100,          // [% of the fundamental wave] (Real Selector: 100-163) 0 => DC component, 1 => fundamental wave, 2=> 2nd harmonic, 3=> 3rd harmonic
    THD_I := 165,                // [-] (Real Selector: 165) "Total Harmonic Distortion" is the distortion factor of the current. It indicates the ratio of the harmonic components of an oscillation relative to its fundamental.
    TDD_I := 166,                // [% of the maximum current] (Real Selector: 166) "Total Demand Distortion" indicates the ratio between the current harmonics and the maximum current (EL3443: 1A and EL3443-0010: 5A)
    RMS_fund_I := 168,           // [A] (Real Selector: 168) Amplitude of the fundamental wave
    F_Ref_I := 169,              // [Hz] (Real Selector: 169) Reference frequency of the current harmonic: Specifies the underlying fundamental frequency, e.g.: 50 or 60 Hz.
    Harmonics_I := 170,          // [% of the fundamental wave] (Real Selector: 170-233) 0 => DC component, 1 => fundamental wave, 2=> 2nd harmonic, 3=> 3rd harmonic
    Error_INDEX_Not_Valid := 255 // [-] (Real Selector: 255) Error message: The selected index is not available.
)UINT;
END_TYPE

// ---- POUs/EL3443/EL3443_DPM/DUTs/E_EL3443_DPM_Total.TcDUT
(*This enum is equivalent to the selectors from the documentation " Confirmation of variable output values 1 - 4"*)
{attribute 'qualified_only'}
TYPE E_EL3443_DPM_Total :
(
    nTotal_OFFSET := 1024,           // Offset for total values. The offset is added to the base selector
    
    In_RMS := 8,                     // [A]  (Real Selector: 1032 (= 1024 + 8))  Calculated RMS value of the neutral current
    Power_Factor := 23,              // [-]  (Real Selector: 1047 (= 1024 + 23))  Total power factor over all phases
    Ptot := 26,                      // [W]  (Real Selector: 1050 (= 1024 + 26))  Total active power
    Ptotavg := 27,                   // [W]  (Real Selector: 1051 (= 1024 + 27))  Average total active power during the last interval
    Ptotmin := 28,                   // [W]  (Real Selector: 1052 (= 1024 + 28))  Minimum total active power in the last interval
    Ptotmax := 29,                   // [W]  (Real Selector: 1053 (= 1024 + 29))  Maximum total active power in the last interval
    Stot := 32,                      // [VA]  (Real Selector: 1056 (= 1024 + 32))  Total apparent power
    Stotavg := 33,                   // [VA]  (Real Selector: 1057 (= 1024 + 33))  Average total apparent power during the last interval
    Stotmin := 34,                   // [VA]  (Real Selector: 1058 (= 1024 + 34))  Minimum total apparent power in the last interval
    Stotmax := 35,                   // [VA]  (Real Selector: 1059 (= 1024 + 35))  Maximum total apparent power in the last interval
    Qtot := 38,                      // [Var]  (Real Selector: 1062 (= 1024 + 38))  Total reactive power
    Qtotavg := 39,                   // [Var]  (Real Selector: 1063 (= 1024 + 39))  Average total reactive power during the last interval
    Qtotmin := 40,                   // [Var]  (Real Selector: 1064 (= 1024 + 40))  Minimum total reactive power in the last interval
    Qtotmax := 41,                   // [Var]  (Real Selector: 1065 (= 1024 + 41))  Maximum total reactive power in the last interval
    Eptot := 45,                     // [mWh]  (ULINT Selector: 1069 (= 1024 + 45))  Balanced total active energy
    EPtot_pos := 46,                 // [mWh]  (ULINT Selector: 1070 (= 1024 + 46))  Related total active energy
    EPtot_neg := 47,                 // [mWh]  (ULINT Selector: 1071 (= 1024 + 47))  Input total active energy
    Eptot_interval := 48,            // [mWh]  (ULINT Selector: 1072 (= 1024 + 48))  Balanced total active energy in last interval
    EPtot_pos_interval := 49,        // [mWh]  (ULINT Selector: 1073 (= 1024 + 49))  Total active energy related in the last interval
    EPtot_neg_interval := 50,        // [mWh]  (ULINT Selector: 1074 (= 1024 + 50))  Input total active energy the last interval
    EStot := 51,                     // [mWh]  (ULINT Selector: 1075 (= 1024 + 51))  Total apparent energy
    EStot_pos := 52,                 // [mWh]  (ULINT Selector: 1076 (= 1024 + 52))  Total apparent energy
    EStot_neg := 53,                 // [mWh]  (ULINT Selector: 1077 (= 1024 + 53))  Total apparent energy
    EStot_interval := 54,            // [mWh]  (ULINT Selector: 1078 (= 1024 + 54))  Total apparent energy in the last interval
    EStot_pos_interval := 55,        // [mWh]  (ULINT Selector: 1079 (= 1024 + 55))  Total apparent energy in the last interval
    EStot_neg_interval := 56,        // [mWh]  (ULINT Selector: 1080 (= 1024 + 56))  Total apparent energy in the last interval
    EQtot := 57,                     // [mWh]  (ULINT Selector: 1081 (= 1024 + 57))  Total reactive energy
    EQtot_pos := 58,                 // [mWh]  (ULINT Selector: 1082 (= 1024 + 58))  Total reactive energy
    EQtot_neg := 59,                 // [mWh]  (ULINT Selector: 1083 (= 1024 + 59))  Total reactive energy
    EQtot_interval := 60,            // [mWh]  (ULINT Selector: 1084 (= 1024 + 60))  Total reactive energy in the last interval
    EQtot_pos_interval := 61,        // [mWh]  (ULINT Selector: 1085 (= 1024 + 61))  Total reactive energy in the last interval
    EQtot_neg_interval := 62,        // [mWh]  (ULINT Selector: 1086 (= 1024 + 62))  Total reactive energy in the last interval
    PhiL1L2 := 70,                   // [°]  (Real Selector: 1094 (= 1024 + 70))  Phase shift angle between phase L1 and L2
    PhiL1L3 := 71,                   // [°]  (Real Selector: 1095 (= 1024 + 71))  Phase shift angle between phase L1 and L3
    Unbalance := 72,                 // [-]  (Real Selector: 1096 (= 1024 + 72))  Ratio between negative and positive voltage system
    PQF := 80,                       // [-]  (Real Selector: 1104 (= 1024 + 80))  Power quality factor
    PQF_Avg := 81,                   // [-]  (Real Selector: 1105 (= 1024 + 81))  Average value of the power quality factor during the last interval
    PQF_MIN := 82,                   // [-]  (Real Selector: 1106 (= 1024 + 82))  Minimum power quality factor in the last interval
    PQF_MAX := 83                    // [-]  (Real Selector: 1107 (= 1024 + 83))  Maximum power quality factor in the last interval
)UINT;      
END_TYPE

// ---- POUs/EL3443/EL3443_DPM/DUTs/ST_EL3443_DPM_MUX_REAL.TcDUT
TYPE ST_EL3443_DPM_MUX_REAL :
STRUCT
    nSelector : UINT := E_EL3443_DPM_Phase.Error_INDEX_Not_Valid;
    fValueRef : REFERENCE TO REAL;
END_STRUCT
END_TYPE

// ---- POUs/EL3443/EL3443_DPM/DUTs/ST_EL3443_DPM_MUX_ULINT.TcDUT
TYPE ST_EL3443_DPM_MUX_ULINT :
STRUCT
    nSelector : UINT := E_EL3443_DPM_Phase.Error_INDEX_Not_Valid;
    nValueRef : POINTER TO ULINT;
END_STRUCT
END_TYPE

// ---- POUs/EL3443/EL3443_DPM/DUTs/ST_EL3443_DPM_StatusLx.TcDUT
TYPE ST_EL3443_DPM_StatusLx :
STRUCT
    bStatus_Voltage_Sign_Bit : BOOL;             //Voltage Sign Bit - Indicates the sign of the current sine wave voltage: 1 = U > 0V, 0 = U < 0V
    bStatus_Overvoltage : BOOL;                  //Overvoltage - Maximum measurable voltage is exceeded.
    bStatus_Overcurrent : BOOL;                  //Overcurrent - Maximum measurable current is exceeded.
    bStatus_Inaccurate_Voltage : BOOL;           //Inaccurate Voltage - The measured voltage value is smaller than the value entered in CoE object "F800:15 Inaccurate Threshold Voltage".
    bStatus_Inaccurate_Current : BOOL;           //Inaccurate Current - The measured current value is smaller than the value entered in CoE object "F800:16 Inaccurate Threshold Current".
    bStatus_Voltage_Guard_Warning : BOOL;        //Voltage Guard Warning - A warning limit of the voltage monitor has been breached.
    bStatus_Voltage_Guard_Error : BOOL;          //Voltage Guard Error - An error limit of the voltage monitor has been breached.
    bStatus_Current_Guard_Warning : BOOL;        //Voltage Current Warning - A warning limit of the Current monitor has been breached.
    bStatus_Current_Guard_Error : BOOL;          //Voltage Current Error - An error limit of the Current monitor has been breached.
    bStatus_TxPDO_Toggle : BOOL;                 //TxPDO Toggle - The TxPDO toggle is toggled by the slave when the data of the associated TxPDO is updated.
END_STRUCT
END_TYPE

// ---- POUs/EL3443/EL3443_DPM/DUTs/ST_EL3443_DPM_StatusTotal.TcDUT
TYPE ST_EL3443_DPM_StatusTotal :
STRUCT
    bStatus_System_State : BOOL;                         //System State - Overall system state (as a logical disjunction of voltage guard errors, phase sequence, overvoltage, overcurrent and frequency guard errors)
    bStatus_Grid_Direction : BOOL;                       //Grid Direction - Phase sequence L1 - L2 - L3 correctly detected (with clockwise 3-phase mains)
    bStatus_Frequency_Guard_Warning : BOOL;              //Frequency Guard Warning - A warning limit of the frequency monitor has been breached.
    bStatus_Frequency_Guard_Error : BOOL;                //Frequency Guard Error - An error limit of the frequency monitor has been breached.
    bStatus_Neutral_Current_Guard_Warning : BOOL;        //Neutral Current Guard Warning - A warning limit of the neutral conductor current monitor has been breached.
    bStatus_Neutral_Current_Guard_Error : BOOL;          //Neutral Current Guard Error - An error limit of the neutral conductor current monitor has been breached.
    bStatus_Active_Power_Guard_Warning : BOOL;           //Active Power Guard Warning - A warning limit of the active power monitor has been breached.
    bStatus_Active_Power_Guard_Error : BOOL;             //Active Power Guard Error - An error limit of the active power monitor has been breached.
    bStatus_Apparent_Power_Guard_Warning : BOOL;         //Apparent Power Guard Warning - A warning limit of the apparent power monitor has been breached.
    bStatus_Apparent_Power_Guard_Error : BOOL;           //Apparent Power Guard Error - An error limit of the apparent power monitor has been breached.
    bStatus_Power_Quality_Guard_Warning : BOOL;          //Power Quality Guard Warning - A warning limit of the PQF monitor has been breached.
    bStatus_Power_Quality_Guard_Error : BOOL;            //Power Quality Guard Error - An error limit of the PQF monitor has been breached.
    bStatus_TxPDO_State : BOOL;                          //TxPDO State - TRUE for general error
    bStatus_TxPDO_Toggle : BOOL;                         //TxPDO Toggle - The TxPDO toggle is toggled by the slave when the data of the associated TxPDO is updated.
    fStatus_Power_Quality_Factor : REAL;                 //Power Quality Factor - Analog value of the voltage quality between 1.0 and 0 (see basic function principles - Power Quality Factor)
END_STRUCT                                              
END_TYPE

// ---- POUs/EL3443/EL3443_DPM/DUTs/ST_EL3443_DPM_VariantLx.TcDUT
TYPE ST_EL3443_DPM_VariantLx :
STRUCT
    fU_RMS : REAL;						// [V] (Real Selector: 1 (Examp.: 257 = 1 + 256 for ch. 1)) RMS value of the voltage
    fU_peak : REAL;						// [V] (Real Selector: 2 (Examp.: 770 = 2 + 768 for ch. 3)) Peak value of the instantaneous voltage in the last interval
    nU_Last_Zero_Cross : ULINT;			// [V] (UINT Selector: 3) DC time of the penultimate voltage zero crossing
    fU_RMS_Minimum : REAL;				// [V] (Real Selector: 4) Minimum RMS value of the voltage in the last interval
    fU_RMS_Maximum : REAL;				// [V] (Real Selector: 5) Maximum RMS value of the voltage in the last interval
    fULL : REAL;						// [V] (Real Selector: 6) RMS value of the phase-to-phase voltage (Channel 1: U_L1L2; Channel 1: U_L2L3; Channel 3: U_L3L1) 
    fI_RMS : REAL;						// [A] (Real Selector: 8) RMS value of the current
    fI_peak : REAL;						// [A] (Real Selector: 9) Peak value of the instantaneous current in the last interval
    fI_RMS_Minimum : REAL;				// [A] (Real Selector: 11) Minimum RMS value of the current in the last interval
    fI_RMS_Maximum : REAL;				// [A] (Real Selector: 12) Maximum RMS value of the current in the last interval
    fFrequency : REAL;					// [Hz] (Real Selector: 17) Frequency of this phase
    fPhi : REAL;						// [°] (Real Selector: 21) Phase angle of the fundamental wave
    fCOS_phi : REAL;					// [-] (Real Selector: 22) Cosine of the fundamental wave phase angle
    fPower_Factor : REAL;				// [-] (Real Selector: 23) Power factor
    fP : REAL;							// [W] (Real Selector: 26) Active power
    fPavg : REAL;						// [W] (Real Selector: 27) Average active power during the last interval
    fPmin : REAL;						// [W] (Real Selector: 28) Minimum active power in the last interval
    fPmax : REAL;						// [W] (Real Selector: 29) Maximum active power in the last interval
    fS : REAL;							// [VA] (Real Selector: 32) Apparent power
    fSavg : REAL;						// [VA] (Real Selector: 33) Average apparent power during the last interval
    fSmin : REAL;						// [VA] (Real Selector: 34) Minimum apparent power in last interval
    fSmax : REAL;						// [VA] (Real Selector: 35) Minimum apparent power in last interval
    fQ : REAL;							// [Var] (Real Selector: 38) Reactive power
    fQavg : REAL;						// [Var] (Real Selector: 39) Average reactive power average during the last interval
    fQmin : REAL;						// [Var] (Real Selector: 40) Minimum reactive power in the last interval
    fQmax : REAL;						// [Var] (Real Selector: 41) Maximum reactive power in the last interval
    nEP : LINT;							// [mhW] (LINT Selector: 45) Recorded active energy
    nEP_pos : ULINT;					// [mhW] (UINT Selector: 46) Received active energy
    nEP_neg : ULINT;					// [mhW] (UINT Selector: 47) Supplied active energy
	nEP_interval : LINT;				// [mhW] (LINT Selector: 48) Recorded active energy in the last interval
	nEP_pos_interval : ULINT;			// [mhW] (UINT Selector: 49) Received active energy in the last interval
	nEP_neg_interval : ULINT;			// [mhW] (UINT Selector: 50) Supplied active energy in the last interval
    nES : LINT;							// [mhW] (LINT Selector: 51) Apparent energy
    nES_pos : ULINT;					// [mhW] (UINT Selector: 52) Apparent energy
    nES_neg : ULINT;					// [mhW] (UINT Selector: 53) Apparent energy
	nES_interval : LINT;				// [mhW] (LINT Selector: 54) Apparent energy in the last interval
	nES_pos_interval : ULINT;			// [mhW] (UINT Selector: 55) Apparent energy in the last interval
	nES_neg_interval : ULINT;			// [mhW] (UINT Selector: 56) Apparent energy in the last interval
    nEQ : LINT;							// [mhW] (LINT Selector: 57) Reactive energy
    nEQ_pos : ULINT;					// [mhW] (UINT Selector: 58) Reactive energy
    nEQ_neg : ULINT;					// [mhW] (UINT Selector: 59) Reactive energy
	nEQ_interval : LINT;				// [mhW] (LINT Selector: 60) Reactive energy in the last interval
	nEQ_pos_interval : ULINT;			// [mhW] (UINT Selector: 62) Reactive energy in the last interval
	nEQ_neg_interval : ULINT;			// [mhW] (UINT Selector: 63) Reactive energy in the last interval
    fTHD_U : REAL;						// [-] (Real Selector: 95) "Total Harmonic Distortion" is the distortion factor of the voltage. It indicates the ratio of the harmonic components of an oscillation relative to its fundamental.
    fRMS_fund_U : REAL;					// [V] (Real Selector: 98) Amplitude of the fundamental wave
    fF_Ref_U : REAL;					// [Hz] (Real Selector: 99) Reference frequency of the voltage harmonic: Specifies the underlying fundamental frequency, e.g.: 50 or 60 Hz.
    fHarmonics_U : ARRAY [0..41] OF REAL;// [% of the fundamental wave] (Real Selector: 100-141) 0 => DC component, 1 => fundamental wave, 2=> 2nd harmonic, 3=> 3rd harmonic
    fTHD_I : REAL;						// [-] (Real Selector: 165) "Total Harmonic Distortion" is the distortion factor of the current. It indicates the ratio of the harmonic components of an oscillation relative to its fundamental.
    fTDD_I : REAL;						// [% of the maximum current] (Real Selector: 166) "Total Demand Distortion" indicates the ratio between the current harmonics and the maximum current (EL3443: 1A and EL3443-0010: 5A)
    fRMS_fund_I : REAL;					// [A] (Real Selector: 168) Amplitude of the fundamental wave
    fF_Ref_I : REAL;					// [Hz] (Real Selector: 169) Reference frequency of the current harmonic: Specifies the underlying fundamental frequency, e.g.: 50 or 60 Hz.
    fHarmonics_I : ARRAY [0..41] OF REAL;// [% of the fundamental wave] (Real Selector: 170-211) 0 => DC component, 1 => fundamental wave, 2=> 2nd harmonic, 3=> 3rd harmonic
END_STRUCT
END_TYPE

// ---- POUs/EL3443/EL3443_DPM/DUTs/ST_EL3443_DPM_VariantTotal.TcDUT
TYPE ST_EL3443_DPM_VariantTotal :
STRUCT
    fIn_RMS : REAL; 			// [A]  (Real Selector: 1032 (= 1024 + 8))  Calculated RMS value of the neutral current
    fPower_Factor : REAL; 		// [-]  (Real Selector: 1047 (= 1024 + 23))  Total power factor over all phases
    fPtot : REAL; 				// [W]  (Real Selector: 1050 (= 1024 + 26))  Total active power
    fPtotavg : REAL; 			// [W]  (Real Selector: 1051 (= 1024 + 27))  Average total active power during the last interval
    fPtotmin : REAL; 			// [W]  (Real Selector: 1052 (= 1024 + 28))  Minimum total active power in the last interval
    fPtotmax : REAL; 			// [W]  (Real Selector: 1053 (= 1024 + 29))  Maximum total active power in the last interval
    fStot : REAL; 				// [VA]  (Real Selector: 1056 (= 1024 + 32))  Total apparent power
    fStotavg : REAL; 			// [VA]  (Real Selector: 1057 (= 1024 + 33))  Average total apparent power during the last interval
    fStotmin : REAL; 			// [VA]  (Real Selector: 1058 (= 1024 + 34))  Minimum total apparent power in the last interval
    fStotmax : REAL; 			// [VA]  (Real Selector: 1059 (= 1024 + 35))  Maximum total apparent power in the last interval
    fQtot : REAL; 				// [Var]  (Real Selector: 1062 (= 1024 + 38))  Total reactive power
    fQtotavg : REAL; 			// [Var]  (Real Selector: 1063 (= 1024 + 39))  Average total reactive power during the last interval
    fQtotmin : REAL; 			// [Var]  (Real Selector: 1064 (= 1024 + 40))  Minimum total reactive power in the last interval
    fQtotmax : REAL; 			// [Var]  (Real Selector: 1065 (= 1024 + 41))  Maximum total reactive power in the last interval
    nEptot : LINT; 				// [mWh]  (LINT Selector: 1069 (= 1024 + 45))  Balanced total active energy
    nEPtot_pos : ULINT; 		// [mWh]  (ULINT Selector: 1070 (= 1024 + 46))  Related total active energy
    nEPtot_neg : ULINT; 		// [mWh]  (ULINT Selector: 1071 (= 1024 + 47))  Input total active energy
    nEptot_interval : LINT; 	// [mWh]  (LINT Selector: 1072 (= 1024 + 48))  Balanced total active energy in last interval
    nEPtot_pos_interval : ULINT;// [mWh]  (ULINT Selector: 1073 (= 1024 + 49))  Total active energy related in the last interval
    nEPtot_neg_interval : ULINT;// [mWh]  (ULINT Selector: 1074 (= 1024 + 50))  Input total active energy the last interval
    nEStot : LINT; 				// [mWh]  (LINT Selector: 1075 (= 1024 + 51))  Total apparent energy
    nEStot_pos : ULINT; 		// [mWh]  (ULINT Selector: 1076 (= 1024 + 52))  Total apparent energy
    nEStot_neg : ULINT; 		// [mWh]  (ULINT Selector: 1077 (= 1024 + 53))  Total apparent energy
    nEStot_interval : LINT; 	// [mWh]  (LINT Selector: 1078 (= 1024 + 54))  Total apparent energy in the last interval
    nEStot_pos_interval : ULINT;// [mWh]  (ULINT Selector: 1079 (= 1024 + 55))  Total apparent energy in the last interval
    nEStot_neg_interval : ULINT;// [mWh]  (ULINT Selector: 1080 (= 1024 + 56))  Total apparent energy in the last interval
    nEQtot : LINT; 				// [mWh]  (LINT Selector: 1081 (= 1024 + 57))  Total reactive energy
    nEQtot_pos : ULINT; 		// [mWh]  (ULINT Selector: 1082 (= 1024 + 58))  Total reactive energy
    nEQtot_neg : ULINT; 		// [mWh]  (ULINT Selector: 1083 (= 1024 + 59))  Total reactive energy
    nEQtot_interval : LINT; 	// [mWh]  (LINT Selector: 1084 (= 1024 + 60))  Total reactive energy in the last interval
    nEQtot_pos_interval : ULINT;// [mWh]  (ULINT Selector: 1085 (= 1024 + 61))  Total reactive energy in the last interval
    nEQtot_neg_interval : ULINT;// [mWh]  (ULINT Selector: 1086 (= 1024 + 62))  Total reactive energy in the last interval
    fPhiL1L2 : REAL; 			// [°]  (Real Selector: 1094 (= 1024 + 70))  Phase shift angle between phase L1 and L2
    fPhiL1L3 : REAL; 			// [°]  (Real Selector: 1095 (= 1024 + 71))  Phase shift angle between phase L1 and L3
    fUnbalance : REAL; 			// [-]  (Real Selector: 1096 (= 1024 + 72))  Ratio between negative and positive voltage system
    fPQF : REAL; 				// [-]  (Real Selector: 1104 (= 1024 + 80))  Power quality factor
    fPQF_Avg : REAL; 			// [-]  (Real Selector: 1105 (= 1024 + 81))  Average value of the power quality factor during the last interval
    fPQF_Min : REAL; 			// [-]  (Real Selector: 1106 (= 1024 + 82))  Minimum power quality factor in the last interval
    fPQF_Max : REAL; 			// [-]  (Real Selector: 1107 (= 1024 + 83))  Maximum power quality factor in the last interval
END_STRUCT
END_TYPE

// ---- POUs/EL3443/EL3443_DPM/DUTs/ST_EL3443_DPM_VariantValues.TcDUT
{attribute 'no-analysis'}
TYPE ST_EL3443_DPM_VariantValues :
STRUCT
	astLx 			: ARRAY[1..3] OF ST_EL3443_DPM_VariantLx;
	stTotal 		: ST_EL3443_DPM_VariantTotal;
END_STRUCT
END_TYPE

// ---- GVLs/GVL_const.TcGVL
{attribute 'qualified_only'}
VAR_GLOBAL
		
	MqttBrokerIPAddress		: STRING		:= '192.168.1.101';
	
	MqttHostPort			: UINT			:= 1883;
	MqttUserName			: STRING		:= 'mqttbroker';
	MqttPassword			: STRING		:= 'IoT-mqttbroker';
	
	LineName 				: STRING		:= 'IoT_Industrial';
	MachineName 			: STRING		:= 'device01';
	
	// PLC diagnostic states
	PlcCpuMemUsage			: STRING		:= 'PlcCpuMemoryUsage';
	PlcCpuCore2Usage		: STRING		:= 'PlcCpuCore2Usage';
	PlcCpuCore3Usage		: STRING		:= 'PlcCpuCore3Usage';
	PlcCpuCore2Jitter		: STRING		:= 'PlcCpuCore2Jitter';
	PlcCpuCore3Jitter		: STRING		:= 'PlcCpuCore3Jitter';
	
	// air flow sensor
	AirFlowSensor			: STRING		:= 'AirFlow1';
	AirPresSensor			: STRING		:= 'AirPressure1';
	AirTempSensor			: STRING		:= 'AirTemperature1';
	
	// ambient temperature & humidity sensor
	AmbientTempSensor		: STRING		:= 'AmbientTemperature';
	AmbientHumiditySensor 	: STRING		:= 'AmbientHumidity';


	// vibration sensors 
	VibSensor1 			:STRING			:= 'Vib1';			
	VibSensor2 			:STRING			:= 'Vib2';			
	VibSensor3 			:STRING			:= 'Vib3';			
	VibSensor4 			:STRING			:= 'Vib4';		
	VibSensor5 			:STRING			:= 'Vib5';			
	VibSensor6 			:STRING			:= 'Vib6';		
	
	// air valves
	AirValve1			:STRING			:= 'AirValve1';
	AirValve2			:STRING			:= 'AirValve2';
	AirValve3			:STRING			:= 'AirValve3';
	AirValve4			:STRING			:= 'AirValve4';
	
	// electrical devices  - periodic operation - (motors/drives)
	ElecDevice1 		: STRING 		:= 'ElecDevice1';
	ElecDevice2 		: STRING 		:= 'ElecDevice2';
	
	// electrical devices  - continous operation 
	ElecDevice3 		: STRING 		:= 'ElecDevice3';
	
	DiffPressSensor1	: STRING		:= 'DiffPressSensor1';
	
END_VAR

// ---- GVLs/GVL_SW.TcGVL
{attribute 'qualified_only'}
VAR_GLOBAL
	
	(*Data FROM and TO Profinet IO-device*)
	PnIoDevice_32Word_In 		: ARRAY[0..31] OF WORD;
	PnIoDevice_32DWord_In 		: ARRAY[0..31] OF DWORD;
	PnIoDevice_10Real_In 		: ARRAY[0..9] OF REAL;
	PnIoDevice_10Real_Out		: ARRAY[0..9] OF REAL;
	
	(* Vibration sensor data *)
	VibSensor1AccelRmsX			: REAL;		
	VibSensor1AccelRmsY			: REAL;
	VibSensor1AccelRmsZ			: REAL;
	VibSensor1Temp				: REAL;
	
	VibSensor2AccelRmsX			: REAL;		
	VibSensor2AccelRmsY			: REAL;
	VibSensor2AccelRmsZ			: REAL;
	VibSensor2Temp				: REAL;
	
	VibSensor3AccelRmsX			: REAL;		
	VibSensor3AccelRmsY			: REAL;
	VibSensor3AccelRmsZ			: REAL;
	VibSensor3Temp				: REAL;
	
	VibSensor4AccelRmsX			: REAL;		 
	VibSensor4AccelRmsY			: REAL;
	VibSensor4AccelRmsZ			: REAL;
	VibSensor4Temp				: REAL;
	
	VibSensor5AccelRmsX			: REAL;		
	VibSensor5AccelRmsY			: REAL;
	VibSensor5AccelRmsZ			: REAL;
	VibSensor5Temp				: REAL;
	
	VibSensor6AccelRmsX			: REAL;		
	VibSensor6AccelRmsY			: REAL;
	VibSensor6AccelRmsZ			: REAL;
	VibSensor6Temp				: REAL;
	
	
	(* Air flow sensor data *)
	AirMassFlowRate				: REAL;			// [kg/h]
	AirFlowVelocity				: REAL;			// [m/s]	
	AirVolume					: REAL;			// [m3]		
	AirVolumetricFlowRate		: REAL;			// [ltr/min]	
	AirMass						: REAL;			// [kg]		
	AirEnergy					: REAL;			// [kWh]	
	AirTemperature				: REAL;			// [°C]		
	AirPressure					: REAL;			// [bar]	
	
	
	(* Ambient environment sensor data *)
	AmbientTempSensor			: REAL;			// [°C]
	AmbientHumiditySensor		: REAL;			// [rel. %]
	
	
	(* Level sensor data *)
	LevelSensor					: REAL;			// [m]
	
	(* Contamination sensor (diff. pressure sensor *)
	DiffPressSensor				: REAL;			// [bar]
	
	
	(* TimeStamp *)
	Unix_TimeStamp 				: ULINT;
		
END_VAR

// ---- GVLs/GVL_HW.TcGVL
{attribute 'qualified_only'}
VAR_GLOBAL
	(* Input Data from Profinet IO-Device*)
	PnIoDevice_32Word_In 			AT%I*: ARRAY[0..31] OF WORD;
	PnIoDevice_32DWord_In 			AT%I*: ARRAY[0..31] OF DWORD;
	PnIoDevice_10Real_In 			AT%I*: ARRAY[0..9] OF REAL;
	
	(* Output Data to Profinet IO-Device*)
	PnIoDevice_10Real_Out 			AT%Q*: ARRAY[0..9] OF REAL;
	
	
	(* Process image data from IO-link node 1 *)  
	IoLinkNode1Ch1_VibAccelRmsX		AT%I*:REAL;
	IoLinkNode1Ch1_VibAccelRmsY		AT%I*:REAL;
	IoLinkNode1Ch1_VibAccelRmsZ		AT%I*:REAL;
	IoLinkNode1Ch1_SensorTemp		AT%I*:REAL;
	
	IoLinkNode1Ch2_VibAccelRmsX		AT%I*:REAL;
	IoLinkNode1Ch2_VibAccelRmsY		AT%I*:REAL;
	IoLinkNode1Ch2_VibAccelRmsZ		AT%I*:REAL;
	IoLinkNode1Ch2_SensorTemp		AT%I*:REAL;
	
	IoLinkNode1Ch3_VibAccelRmsX		AT%I*:REAL;
	IoLinkNode1Ch3_VibAccelRmsY		AT%I*:REAL;
	IoLinkNode1Ch3_VibAccelRmsZ		AT%I*:REAL;
	IoLinkNode1Ch3_SensorTemp		AT%I*:REAL;
	
	IoLinkNode1Ch4_VibAccelRmsX		AT%I*:REAL;
	IoLinkNode1Ch4_VibAccelRmsY		AT%I*:REAL;
	IoLinkNode1Ch4_VibAccelRmsZ		AT%I*:REAL;
	IoLinkNode1Ch4_SensorTemp		AT%I*:REAL;
	
	IoLinkNode1Ch5_VibAccelRmsX		AT%I*:REAL;
	IoLinkNode1Ch5_VibAccelRmsY		AT%I*:REAL;
	IoLinkNode1Ch5_VibAccelRmsZ		AT%I*:REAL;
	IoLinkNode1Ch5_SensorTemp		AT%I*:REAL;
	
	IoLinkNode1Ch6_VibAccelRmsX		AT%I*:REAL;
	IoLinkNode1Ch6_VibAccelRmsY		AT%I*:REAL;
	IoLinkNode1Ch6_VibAccelRmsZ		AT%I*:REAL;
	IoLinkNode1Ch6_SensorTemp		AT%I*:REAL;
	
	(* Process image data from IO-link node 2 *)
	IoLinkNode2Ch1_MassFlowRate		AT%I*:REAL;		// [kg/h]
	IoLinkNode2Ch1_FlowVelocity		AT%I*:REAL;		// [m/s]
	IoLinkNode2Ch1_Volume			AT%I*:REAL;		// [m3]
	IoLinkNode2Ch1_VolFlowRate		AT%I*:REAL;		// [m3/h]
	IoLinkNode2Ch1_Mass				AT%I*:REAL;		// [kg]
	IoLinkNode2Ch1_Energy			AT%I*:REAL;		// [kWh]
	IoLinkNode2Ch1_Temperature		AT%I*:REAL;		// [°C]	
	IoLinkNode2Ch1_Pressure			AT%I*:REAL;		// [bar]
	
	IoLinkNode2Ch2_Temperature		AT%I*: ARRAY[1..2] OF USINT;
	IoLinkNode2Ch2_Humidity			AT%I*: ARRAY[1..2] OF USINT;
	
	IoLinkNode2Ch3_Level			AT%I*: INT;		// [m] * 0.001
	
	IoLinkNode2Ch4_DiffPress		AT%I*: UINT;	// [bar] * 0.1	
	
	
END_VAR

// ---- GVLs/GVL_Visu.TcGVL
{attribute 'qualified_only'}
VAR_GLOBAL
		
	ButtonStart 			: BOOL;
	LineRunning				: BOOL;
	LineProducing			: BOOL;
	LineSpeed				: UINT := 50;
	
